LIN {X 0,Y 196.007,Z 648.874,A -85,B 0,C 180,E1 -19663.155,E2 -19663.155} C_VEL
LIN {X 0,Y 201.591,Z 629.624,A -85,B 0,C 180,E1 -19666.019,E2 -19666.019} C_VEL
LIN {X 0,Y 207.04,Z 608.516,A -85,B 0,C 180,E1 -19668.466,E2 -19668.466} C_VEL
LIN {X 0,Y 211.706,Z 587.34,A -85,B 0,C 180,E1 -19670.34,E2 -19670.34} C_VEL
LIN {X 0,Y 215.64,Z 565.396,A -85,B 0,C 180,E1 -19671.754,E2 -19671.754} C_VEL
LIN {X 0,Y 234.928,Z 427.617,A -85,B 0,C 180,E1 -19677.857,E2 -19677.857} C_VEL
LIN {X 0,Y 233.125,Z 424.133,A -85,B 0,C 180,E1 -19678.519,E2 -19678.519} C_VEL
LIN {X 0,Y 230.769,Z 425.807,A -85,B 0,C 180,E1 -19678.936,E2 -19678.936} C_VEL
LIN {X 0,Y 225.246,Z 433.176,A -85,B 0,C 180,E1 -19679.67,E2 -19679.67} C_VEL
LIN {X 0,Y 221.567,Z 436.319,A -85,B 0,C 180,E1 -19680.31,E2 -19680.31} C_VEL
LIN {X 0,Y 219.541,Z 437.961,A -85,B 0,C 180,E1 -19680.833,E2 -19680.833} C_VEL
LIN {X 0,Y 218.156,Z 442.528,A -85,B 0,C 180,E1 -19681.53,E2 -19681.53} C_VEL
LIN {X 0,Y 209.499,Z 487.735,A -85,B 0,C 180,E1 -19687.301,E2 -19687.301} C_VEL
LIN {X 0,Y 210.664,Z 518.818,A -85,B 0,C 180,E1 -19689.081,E2 -19689.081} C_VEL
LIN {X 0,Y 202.963,Z 633.554,A -85,B 0,C 180,E1 -19692.805,E2 -19692.805} C_VEL
LIN {X 0,Y 200.899,Z 650.257,A -85,B 0,C 180,E1 -19693.856,E2 -19693.856} C_VEL
LIN {X 0,Y 198.235,Z 665.159,A -85,B 0,C 180,E1 -19695.24,E2 -19695.24} C_VEL
LIN {X 0,Y 194.818,Z 679.656,A -85,B 0,C 180,E1 -19697.097,E2 -19697.097} C_VEL
LIN {X 0,Y 190.653,Z 694.187,A -85,B 0,C 180,E1 -19699.573,E2 -19699.573} C_VEL
LIN {X 0,Y 186.361,Z 706.922,A -85,B 0,C 180,E1 -19702.444,E2 -19702.444} C_VEL
LIN {X 0,Y 181.968,Z 718.732,A -85,B 0,C 180,E1 -19705.9,E2 -19705.9} C_VEL
LIN {X 0,Y 177.982,Z 728.651,A -85,B 0,C 180,E1 -19709.691,E2 -19709.691} C_VEL
LIN {X 0,Y 174.23,Z 737.787,A -85,B 0,C 180,E1 -19714.275,E2 -19714.275} C_VEL
LIN {X 0,Y 171.426,Z 744.822,A -85,B 0,C 180,E1 -19719.057,E2 -19719.057} C_VEL
LIN {X 0,Y 169.483,Z 750.379,A -85,B 0,C 180,E1 -19724.342,E2 -19724.342} C_VEL
LIN {X 0,Y 168.571,Z 753.881,A -85,B 0,C 180,E1 -19729.419,E2 -19729.419} C_VEL
LIN {X 0,Y 168.319,Z 755.89,A -85,B 0,C 180,E1 -19734.941,E2 -19734.941} C_VEL
LIN {X 0,Y 168.642,Z 756.21,A -85,B 0,C 180,E1 -19740.257,E2 -19740.257} C_VEL
LIN {X 0,Y 169.762,Z 754.819,A -85,B 0,C 180,E1 -19745.663,E2 -19745.663} C_VEL
LIN {X 0,Y 172.008,Z 751.682,A -85,B 0,C 180,E1 -19751.055,E2 -19751.055} C_VEL
LIN {X 0,Y 175.241,Z 747.035,A -85,B 0,C 180,E1 -19755.959,E2 -19755.959} C_VEL
LIN {X 0,Y 179.593,Z 740.487,A -85,B 0,C 180,E1 -19760.696,E2 -19760.696} C_VEL
LIN {X 0,Y 184.754,Z 732.288,A -85,B 0,C 180,E1 -19764.993,E2 -19764.993} C_VEL
LIN {X 0,Y 190.458,Z 722.323,A -85,B 0,C 180,E1 -19768.831,E2 -19768.831} C_VEL
LIN {X 0,Y 196.127,Z 711.358,A -85,B 0,C 180,E1 -19772.028,E2 -19772.028} C_VEL
LIN {X 0,Y 201.673,Z 698.951,A -85,B 0,C 180,E1 -19774.761,E2 -19774.761} C_VEL
LIN {X 0,Y 206.822,Z 685.498,A -85,B 0,C 180,E1 -19777.021,E2 -19777.021} C_VEL
LIN {X 0,Y 211.423,Z 670.576,A -85,B 0,C 180,E1 -19778.882,E2 -19778.882} C_VEL
LIN {X 0,Y 214.892,Z 656.116,A -85,B 0,C 180,E1 -19780.217,E2 -19780.217} C_VEL
LIN {X 0,Y 217.57,Z 640.183,A -85,B 0,C 180,E1 -19781.237,E2 -19781.237} C_VEL
LIN {X 0,Y 219.391,Z 621.388,A -85,B 0,C 180,E1 -19781.962,E2 -19781.962} C_VEL
LIN {X 0,Y 227.565,Z 519.665,A -85,B 0,C 180,E1 -19784.999,E2 -19784.999} C_VEL
LIN {X 0,Y 226.964,Z 491.665,A -85,B 0,C 180,E1 -19787.015,E2 -19787.015} C_VEL
LIN {X 0,Y 227.705,Z 486.476,A -85,B 0,C 180,E1 -19787.574,E2 -19787.574} C_VEL
LIN {X 0,Y 238.01,Z 442.856,A -85,B 0,C 180,E1 -19792.88,E2 -19792.88} C_VEL
LIN {X 0,Y 238.558,Z 440.651,A -85,B 0,C 180,E1 -19793.146,E2 -19793.146} C_VEL
LIN {X 0,Y 239.044,Z 437.189,A -85,B 0,C 180,E1 -19793.775,E2 -19793.775} C_VEL
LIN {X 0,Y 238.564,Z 433.691,A -85,B 0,C 180,E1 -19794.923,E2 -19794.923} C_VEL
LIN {X 0,Y 236.422,Z 427.479,A -85,B 0,C 180,E1 -19797.96,E2 -19797.96} C_VEL
LIN {X 0,Y 235.366,Z 419.825,A -85,B 0,C 180,E1 -19801.46,E2 -19801.46} C_VEL
LIN {X 0,Y 234.261,Z 414.19,A -85,B 0,C 180,E1 -19804.896,E2 -19804.896} C_VEL
LIN {X 0,Y 233.64,Z 409.636,A -85,B 0,C 180,E1 -19808.698,E2 -19808.698} C_VEL
LIN {X 0,Y 233.642,Z 406.373,A -85,B 0,C 180,E1 -19813.36,E2 -19813.36} C_VEL
LIN {X 0,Y 233.888,Z 406.188,A -85,B 0,C 180,E1 -19817.411,E2 -19817.411} C_VEL
LIN {X 0,Y 233.923,Z 406.605,A -85,B 0,C 180,E1 -19817.923,E2 -19817.923} C_VEL
LIN {X 0,Y 231.401,Z 422.323,A -85,B 0,C 180,E1 -19823.656,E2 -19823.656} C_VEL
LIN {X 0,Y 231.464,Z 426.766,A -85,B 0,C 180,E1 -19825.164,E2 -19825.164} C_VEL
LIN {X 0,Y 234.206,Z 432.58,A -85,B 0,C 180,E1 -19826.234,E2 -19826.234} C_VEL
LIN {X 0,Y 214.117,Z 574.365,A -85,B 0,C 180,E1 -19832.298,E2 -19832.298} C_VEL
LIN {X 0,Y 209.776,Z 596.826,A -85,B 0,C 180,E1 -19833.73,E2 -19833.73} C_VEL
LIN {X 0,Y 204.359,Z 619.531,A -85,B 0,C 180,E1 -19835.697,E2 -19835.697} C_VEL
LIN {X 0,Y 203.513,Z 624.212,A -85,B 0,C 180,E1 -19836.005,E2 -19836.005} C_VEL
LIN {X 0,Y 201.91,Z 648.108,A -85,B 0,C 180,E1 -19837.239,E2 -19837.239} C_VEL
LIN {X 0,Y 200,Z 662.648,A -85,B 0,C 180,E1 -19838.353,E2 -19838.353} C_VEL
LIN {X 0,Y 197.204,Z 676.915,A -85,B 0,C 180,E1 -19839.82,E2 -19839.82} C_VEL
LIN {X 0,Y 193.529,Z 691.091,A -85,B 0,C 180,E1 -19841.713,E2 -19841.713} C_VEL
LIN {X 0,Y 188.844,Z 705.51,A -85,B 0,C 180,E1 -19844.24,E2 -19844.24} C_VEL
LIN {X 0,Y 183.859,Z 718.529,A -85,B 0,C 180,E1 -19847.18,E2 -19847.18} C_VEL
LIN {X 0,Y 178.555,Z 730.688,A -85,B 0,C 180,E1 -19850.75,E2 -19850.75} C_VEL
LIN {X 0,Y 173.494,Z 741.383,A -85,B 0,C 180,E1 -19854.814,E2 -19854.814} C_VEL
LIN {X 0,Y 168.92,Z 750.58,A -85,B 0,C 180,E1 -19859.404,E2 -19859.404} C_VEL
LIN {X 0,Y 164.889,Z 758.8,A -85,B 0,C 180,E1 -19864.888,E2 -19864.888} C_VEL
LIN {X 0,Y 162.145,Z 764.84,A -85,B 0,C 180,E1 -19870.554,E2 -19870.554} C_VEL
LIN {X 0,Y 160.629,Z 769.021,A -85,B 0,C 180,E1 -19876.322,E2 -19876.322} C_VEL
LIN {X 0,Y 160.192,Z 771.404,A -85,B 0,C 180,E1 -19882.111,E2 -19882.111} C_VEL
LIN {X 0,Y 160.319,Z 772.033,A -85,B 0,C 180,E1 -19887.502,E2 -19887.502} C_VEL
LIN {X 0,Y 160.369,Z 771.303,A -85,B 0,C 180,E1 -19892.148,E2 -19892.148} C_VEL
LIN {X 0,Y 160.352,Z 768.92,A -85,B 0,C 180,E1 -19897.888,E2 -19897.888} C_VEL
LIN {X 0,Y 160.947,Z 769.601,A -85,B 0,C 180,E1 -19905.497,E2 -19905.497} C_VEL
LIN {X 0,Y 164.172,Z 768.537,A -85,B 0,C 180,E1 -19913.705,E2 -19913.705} C_VEL
LIN {X 0,Y 171.188,Z 765.587,A -85,B 0,C 180,E1 -19922.126,E2 -19922.126} C_VEL
LIN {X 0,Y 183.295,Z 760.405,A -85,B 0,C 180,E1 -19930.48,E2 -19930.48} C_VEL
LIN {X 0,Y 199.447,Z 753.565,A -85,B 0,C 180,E1 -19937.475,E2 -19937.475} C_VEL
LIN {X 0,Y 201.156,Z 752.825,A -85,B 0,C 180,E1 -19938.142,E2 -19938.142} C_VEL
LIN {X 0,Y 185.881,Z 756.616,A -85,B 0,C 180,E1 -19944.485,E2 -19944.485} C_VEL
LIN {X 0,Y 174.097,Z 758.634,A -85,B 0,C 180,E1 -19951.906,E2 -19951.906} C_VEL
LIN {X 0,Y 166.488,Z 758.702,A -85,B 0,C 180,E1 -19959.616,E2 -19959.616} C_VEL
LIN {X 0,Y 162.328,Z 757.034,A -85,B 0,C 180,E1 -19967.19,E2 -19967.19} C_VEL
LIN {X 0,Y 160.621,Z 753.914,A -85,B 0,C 180,E1 -19974.285,E2 -19974.285} C_VEL
LIN {X 0,Y 160.227,Z 749.933,A -85,B 0,C 180,E1 -19980.359,E2 -19980.359} C_VEL
LIN {X 0,Y 160.288,Z 744.773,A -85,B 0,C 180,E1 -19986.089,E2 -19986.089} C_VEL
LIN {X 0,Y 161.003,Z 737.672,A -85,B 0,C 180,E1 -19992.191,E2 -19992.191} C_VEL
LIN {X 0,Y 162.736,Z 728.688,A -85,B 0,C 180,E1 -19998.262,E2 -19998.262} C_VEL
LIN {X 0,Y 165.518,Z 718.279,A -85,B 0,C 180,E1 -20003.876,E2 -20003.876} C_VEL
LIN {X 0,Y 169.491,Z 705.708,A -85,B 0,C 180,E1 -20009.318,E2 -20009.318} C_VEL
LIN {X 0,Y 174.318,Z 691.587,A -85,B 0,C 180,E1 -20014.204,E2 -20014.204} C_VEL
LIN {X 0,Y 179.96,Z 675.353,A -85,B 0,C 180,E1 -20018.688,E2 -20018.688} C_VEL
LIN {X 0,Y 185.561,Z 658.707,A -85,B 0,C 180,E1 -20022.342,E2 -20022.342} C_VEL
LIN {X 0,Y 191.569,Z 639.598,A -85,B 0,C 180,E1 -20025.649,E2 -20025.649} C_VEL
LIN {X 0,Y 197.398,Z 619.056,A -85,B 0,C 180,E1 -20028.426,E2 -20028.426} C_VEL
LIN {X 0,Y 202.545,Z 598.322,A -85,B 0,C 180,E1 -20030.586,E2 -20030.586} C_VEL
LIN {X 0,Y 207.089,Z 576.326,A -85,B 0,C 180,E1 -20032.301,E2 -20032.301} C_VEL
LIN {X 0,Y 211.001,Z 551.851,A -85,B 0,C 180,E1 -20033.646,E2 -20033.646} C_VEL
LIN {X 0,Y 227.233,Z 440.079,A -85,B 0,C 180,E1 -20038.675,E2 -20038.675} C_VEL
LIN {X 0,Y 222.58,Z 443.633,A -85,B 0,C 180,E1 -20039.492,E2 -20039.492} C_VEL
LIN {X 0,Y 221.414,Z 444.853,A -85,B 0,C 180,E1 -20039.67,E2 -20039.67} C_VEL
LIN {X 0,Y 216.084,Z 451.918,A -85,B 0,C 180,E1 -20040.389,E2 -20040.389} C_VEL
LIN {X 0,Y 212.316,Z 455.133,A -85,B 0,C 180,E1 -20041.058,E2 -20041.058} C_VEL
LIN {X 0,Y 210.266,Z 456.816,A -85,B 0,C 180,E1 -20041.604,E2 -20041.604} C_VEL
LIN {X 0,Y 208.844,Z 461.49,A -85,B 0,C 180,E1 -20042.326,E2 -20042.326} C_VEL
LIN {X 0,Y 203.614,Z 488.758,A -85,B 0,C 180,E1 -20045.822,E2 -20045.822} C_VEL
LIN {X 0,Y 204.632,Z 519.551,A -85,B 0,C 180,E1 -20047.637,E2 -20047.637} C_VEL
LIN {X 0,Y 196.623,Z 633.934,A -85,B 0,C 180,E1 -20051.409,E2 -20051.409} C_VEL
LIN {X 0,Y 194.482,Z 650.561,A -85,B 0,C 180,E1 -20052.475,E2 -20052.475} C_VEL
LIN {X 0,Y 191.599,Z 665.988,A -85,B 0,C 180,E1 -20053.941,E2 -20053.941} C_VEL
LIN {X 0,Y 187.788,Z 681.269,A -85,B 0,C 180,E1 -20055.977,E2 -20055.977} C_VEL
LIN {X 0,Y 183.461,Z 695.537,A -85,B 0,C 180,E1 -20058.523,E2 -20058.523} C_VEL
LIN {X 0,Y 178.786,Z 708.651,A -85,B 0,C 180,E1 -20061.636,E2 -20061.636} C_VEL
LIN {X 0,Y 174.426,Z 719.757,A -85,B 0,C 180,E1 -20065.064,E2 -20065.064} C_VEL
LIN {X 0,Y 169.976,Z 730.229,A -85,B 0,C 180,E1 -20069.322,E2 -20069.322} C_VEL
LIN {X 0,Y 166.35,Z 738.634,A -85,B 0,C 180,E1 -20073.816,E2 -20073.816} C_VEL
LIN {X 0,Y 163.459,Z 745.511,A -85,B 0,C 180,E1 -20078.792,E2 -20078.792} C_VEL
LIN {X 0,Y 161.462,Z 750.998,A -85,B 0,C 180,E1 -20084.337,E2 -20084.337} C_VEL
LIN {X 0,Y 160.513,Z 754.566,A -85,B 0,C 180,E1 -20090.031,E2 -20090.031} C_VEL
LIN {X 0,Y 160.333,Z 756.348,A -85,B 0,C 180,E1 -20095.482,E2 -20095.482} C_VEL
LIN {X 0,Y 160.754,Z 756.579,A -85,B 0,C 180,E1 -20101.076,E2 -20101.076} C_VEL
LIN {X 0,Y 162.224,Z 754.933,A -85,B 0,C 180,E1 -20107.153,E2 -20107.153} C_VEL
LIN {X 0,Y 164.898,Z 751.567,A -85,B 0,C 180,E1 -20112.802,E2 -20112.802} C_VEL
LIN {X 0,Y 168.893,Z 746.228,A -85,B 0,C 180,E1 -20118.232,E2 -20118.232} C_VEL
LIN {X 0,Y 173.835,Z 739.315,A -85,B 0,C 180,E1 -20123.075,E2 -20123.075} C_VEL
LIN {X 0,Y 179.748,Z 730.328,A -85,B 0,C 180,E1 -20127.556,E2 -20127.556} C_VEL
LIN {X 0,Y 185.805,Z 720.142,A -85,B 0,C 180,E1 -20131.291,E2 -20131.291} C_VEL
LIN {X 0,Y 192.09,Z 708.2,A -85,B 0,C 180,E1 -20134.56,E2 -20134.56} C_VEL
LIN {X 0,Y 197.59,Z 696.12,A -85,B 0,C 180,E1 -20137.067,E2 -20137.067} C_VEL
LIN {X 0,Y 203.058,Z 681.742,A -85,B 0,C 180,E1 -20139.308,E2 -20139.308} C_VEL
LIN {X 0,Y 207.513,Z 667.094,A -85,B 0,C 180,E1 -20141.001,E2 -20141.001} C_VEL
LIN {X 0,Y 211.23,Z 650.563,A -85,B 0,C 180,E1 -20142.364,E2 -20142.364} C_VEL
LIN {X 0,Y 213.59,Z 634.571,A -85,B 0,C 180,E1 -20143.234,E2 -20143.234} C_VEL
LIN {X 0,Y 223.224,Z 520.734,A -85,B 0,C 180,E1 -20146.695,E2 -20146.695} C_VEL
LIN {X 0,Y 222.906,Z 493.056,A -85,B 0,C 180,E1 -20148.747,E2 -20148.747} C_VEL
LIN {X 0,Y 223.234,Z 488.794,A -85,B 0,C 180,E1 -20149.156,E2 -20149.156} C_VEL
LIN {X 0,Y 233.54,Z 447.232,A -85,B 0,C 180,E1 -20154.225,E2 -20154.225} C_VEL
LIN {X 0,Y 237.089,Z 432.81,A -85,B 0,C 180,E1 -20156.009,E2 -20156.009} C_VEL
LIN {X 0,Y 236.422,Z 427.479,A -85,B 0,C 180,E1 -20157.96,E2 -20157.96} C_VEL
LIN {X 0,Y 235.623,Z 424.837,A -85,B 0,C 180,E1 -20159.425,E2 -20159.425} C_VEL
LIN {X 0,Y 233.667,Z 422.928,A -85,B 0,C 180,E1 -20161.79,E2 -20161.79} C_VEL
LIN {X 0,Y 231.182,Z 421.007,A -85,B 0,C 180,E1 -20165.355,E2 -20165.355} C_VEL
LIN {X 0,Y 230.926,Z 419.801,A -85,B 0,C 180,E1 -20166.437,E2 -20166.437} C_VEL
LIN {X 0,Y 230.46,Z 416.606,A -85,B 0,C 180,E1 -20169.488,E2 -20169.488} C_VEL
LIN {X 0,Y 230.78,Z 413.806,A -85,B 0,C 180,E1 -20173.785,E2 -20173.785} C_VEL
LIN {X 0,Y 231.018,Z 413.815,A -85,B 0,C 180,E1 -20177.245,E2 -20177.245} C_VEL
LIN {X 0,Y 228.173,Z 430.939,A -85,B 0,C 180,E1 -20183.5,E2 -20183.5} C_VEL
LIN {X 0,Y 228.012,Z 435.468,A -85,B 0,C 180,E1 -20184.971,E2 -20184.971} C_VEL
LIN {X 0,Y 207.408,Z 574.805,A -85,B 0,C 180,E1 -20191.105,E2 -20191.105} C_VEL
LIN {X 0,Y 202.897,Z 597.264,A -85,B 0,C 180,E1 -20192.583,E2 -20192.583} C_VEL
LIN {X 0,Y 201.248,Z 605.535,A -85,B 0,C 180,E1 -20193.136,E2 -20193.136} C_VEL
LIN {X 0,Y 200.055,Z 621.802,A -85,B 0,C 180,E1 -20193.871,E2 -20193.871} C_VEL
LIN {X 0,Y 199.017,Z 637.587,A -85,B 0,C 180,E1 -20194.64,E2 -20194.64} C_VEL
LIN {X 0,Y 197.793,Z 650.252,A -85,B 0,C 180,E1 -20195.36,E2 -20195.36} C_VEL
LIN {X 0,Y 195.668,Z 663.933,A -85,B 0,C 180,E1 -20196.44,E2 -20196.44} C_VEL
LIN {X 0,Y 192.609,Z 677.955,A -85,B 0,C 180,E1 -20197.909,E2 -20197.909} C_VEL
LIN {X 0,Y 188.65,Z 691.693,A -85,B 0,C 180,E1 -20199.786,E2 -20199.786} C_VEL
LIN {X 0,Y 183.485,Z 706.278,A -85,B 0,C 180,E1 -20202.398,E2 -20202.398} C_VEL
LIN {X 0,Y 178.044,Z 719.249,A -85,B 0,C 180,E1 -20205.42,E2 -20205.42} C_VEL
LIN {X 0,Y 172.357,Z 731.173,A -85,B 0,C 180,E1 -20209.046,E2 -20209.046} C_VEL
LIN {X 0,Y 166.901,Z 741.673,A -85,B 0,C 180,E1 -20213.202,E2 -20213.202} C_VEL
LIN {X 0,Y 161.621,Z 751.27,A -85,B 0,C 180,E1 -20218.28,E2 -20218.28} C_VEL
LIN {X 0,Y 157.511,Z 758.77,A -85,B 0,C 180,E1 -20223.623,E2 -20223.623} C_VEL
LIN {X 0,Y 154.463,Z 764.695,A -85,B 0,C 180,E1 -20229.545,E2 -20229.545} C_VEL
LIN {X 0,Y 152.725,Z 768.827,A -85,B 0,C 180,E1 -20235.674,E2 -20235.674} C_VEL
LIN {X 0,Y 152.201,Z 771.06,A -85,B 0,C 180,E1 -20241.694,E2 -20241.694} C_VEL
LIN {X 0,Y 152.323,Z 771.623,A -85,B 0,C 180,E1 -20247.371,E2 -20247.371} C_VEL
LIN {X 0,Y 152.378,Z 770.824,A -85,B 0,C 180,E1 -20252.26,E2 -20252.26} C_VEL
LIN {X 0,Y 152.369,Z 768.382,A -85,B 0,C 180,E1 -20257.925,E2 -20257.925} C_VEL
LIN {X 0,Y 152.403,Z 768.051,A -85,B 0,C 180,E1 -20259.063,E2 -20259.063} C_VEL
LIN {X 0,Y 153.327,Z 768.816,A -85,B 0,C 180,E1 -20267.069,E2 -20267.069} C_VEL
LIN {X 0,Y 157.422,Z 767.916,A -85,B 0,C 180,E1 -20275.996,E2 -20275.996} C_VEL
LIN {X 0,Y 166.294,Z 764.952,A -85,B 0,C 180,E1 -20285.259,E2 -20285.259} C_VEL
LIN {X 0,Y 179.981,Z 760.058,A -85,B 0,C 180,E1 -20293.544,E2 -20293.544} C_VEL
LIN {X 0,Y 190.979,Z 756.033,A -85,B 0,C 180,E1 -20298.205,E2 -20298.205} C_VEL
LIN {X 0,Y 175.669,Z 758.775,A -85,B 0,C 180,E1 -20305.051,E2 -20305.051} C_VEL
LIN {X 0,Y 164.759,Z 759.68,A -85,B 0,C 180,E1 -20312.536,E2 -20312.536} C_VEL
LIN {X 0,Y 157.483,Z 758.803,A -85,B 0,C 180,E1 -20320.724,E2 -20320.724} C_VEL
LIN {X 0,Y 153.749,Z 756.259,A -85,B 0,C 180,E1 -20328.751,E2 -20328.751} C_VEL
LIN {X 0,Y 152.428,Z 752.31,A -85,B 0,C 180,E1 -20336.24,E2 -20336.24} C_VEL
LIN {X 0,Y 152.211,Z 747.873,A -85,B 0,C 180,E1 -20342.26,E2 -20342.26} C_VEL
LIN {X 0,Y 152.462,Z 741.959,A -85,B 0,C 180,E1 -20348.297,E2 -20348.297} C_VEL
LIN {X 0,Y 153.556,Z 733.994,A -85,B 0,C 180,E1 -20354.712,E2 -20354.712} C_VEL
LIN {X 0,Y 155.863,Z 724.042,A -85,B 0,C 180,E1 -20361.055,E2 -20361.055} C_VEL
LIN {X 0,Y 159.422,Z 712.205,A -85,B 0,C 180,E1 -20367.045,E2 -20367.045} C_VEL
LIN {X 0,Y 164.001,Z 698.806,A -85,B 0,C 180,E1 -20372.448,E2 -20372.448} C_VEL
LIN {X 0,Y 169.34,Z 683.884,A -85,B 0,C 180,E1 -20377.245,E2 -20377.245} C_VEL
LIN {X 0,Y 175.192,Z 667.429,A -85,B 0,C 180,E1 -20381.457,E2 -20381.457} C_VEL
LIN {X 0,Y 181.263,Z 649.43,A -85,B 0,C 180,E1 -20385.081,E2 -20385.081} C_VEL
LIN {X 0,Y 187.216,Z 630.282,A -85,B 0,C 180,E1 -20388.116,E2 -20388.116} C_VEL
LIN {X 0,Y 193.011,Z 609.33,A -85,B 0,C 180,E1 -20390.692,E2 -20390.692} C_VEL
LIN {X 0,Y 198.029,Z 588.042,A -85,B 0,C 180,E1 -20392.679,E2 -20392.679} C_VEL
LIN {X 0,Y 202.33,Z 565.771,A -85,B 0,C 180,E1 -20394.195,E2 -20394.195} C_VEL
LIN {X 0,Y 218.439,Z 458.466,A -85,B 0,C 180,E1 -20399.293,E2 -20399.293} C_VEL
LIN {X 0,Y 213.978,Z 462.059,A -85,B 0,C 180,E1 -20400.076,E2 -20400.076} C_VEL
LIN {X 0,Y 212.508,Z 463.195,A -85,B 0,C 180,E1 -20400.339,E2 -20400.339} C_VEL
LIN {X 0,Y 207.004,Z 470.589,A -85,B 0,C 180,E1 -20401.075,E2 -20401.075} C_VEL
LIN {X 0,Y 203.137,Z 473.924,A -85,B 0,C 180,E1 -20401.772,E2 -20401.772} C_VEL
LIN {X 0,Y 201.131,Z 475.381,A -85,B 0,C 180,E1 -20402.299,E2 -20402.299} C_VEL
LIN {X 0,Y 199.828,Z 478.864,A -85,B 0,C 180,E1 -20402.911,E2 -20402.911} C_VEL
LIN {X 0,Y 197.861,Z 489.188,A -85,B 0,C 180,E1 -20404.218,E2 -20404.218} C_VEL
LIN {X 0,Y 198.705,Z 520.426,A -85,B 0,C 180,E1 -20406.116,E2 -20406.116} C_VEL
LIN {X 0,Y 190.39,Z 634.283,A -85,B 0,C 180,E1 -20409.927,E2 -20409.927} C_VEL
LIN {X 0,Y 188.148,Z 650.98,A -85,B 0,C 180,E1 -20411.015,E2 -20411.015} C_VEL
LIN {X 0,Y 185.065,Z 666.733,A -85,B 0,C 180,E1 -20412.548,E2 -20412.548} C_VEL
LIN {X 0,Y 181.093,Z 681.937,A -85,B 0,C 180,E1 -20414.628,E2 -20414.628} C_VEL
LIN {X 0,Y 176.819,Z 695.455,A -85,B 0,C 180,E1 -20417.09,E2 -20417.09} C_VEL
LIN {X 0,Y 171.909,Z 708.656,A -85,B 0,C 180,E1 -20420.286,E2 -20420.286} C_VEL
LIN {X 0,Y 167.314,Z 719.842,A -85,B 0,C 180,E1 -20423.821,E2 -20423.821} C_VEL
LIN {X 0,Y 162.608,Z 730.379,A -85,B 0,C 180,E1 -20428.234,E2 -20428.234} C_VEL
LIN {X 0,Y 158.779,Z 738.788,A -85,B 0,C 180,E1 -20432.884,E2 -20432.884} C_VEL
LIN {X 0,Y 155.602,Z 745.937,A -85,B 0,C 180,E1 -20438.274,E2 -20438.274} C_VEL
LIN {X 0,Y 153.529,Z 751.319,A -85,B 0,C 180,E1 -20443.977,E2 -20443.977} C_VEL
LIN {X 0,Y 152.525,Z 754.902,A -85,B 0,C 180,E1 -20449.926,E2 -20449.926} C_VEL
LIN {X 0,Y 152.349,Z 756.776,A -85,B 0,C 180,E1 -20455.954,E2 -20455.954} C_VEL
LIN {X 0,Y 152.859,Z 756.971,A -85,B 0,C 180,E1 -20461.749,E2 -20461.749} C_VEL
LIN {X 0,Y 154.466,Z 755.389,A -85,B 0,C 180,E1 -20467.942,E2 -20467.942} C_VEL
LIN {X 0,Y 157.379,Z 752.102,A -85,B 0,C 180,E1 -20473.822,E2 -20473.822} C_VEL
LIN {X 0,Y 161.744,Z 746.766,A -85,B 0,C 180,E1 -20479.526,E2 -20479.526} C_VEL
LIN {X 0,Y 167.015,Z 739.953,A -85,B 0,C 180,E1 -20484.499,E2 -20484.499} C_VEL
LIN {X 0,Y 173.311,Z 731.031,A -85,B 0,C 180,E1 -20489.104,E2 -20489.104} C_VEL
LIN {X 0,Y 179.697,Z 721.022,A -85,B 0,C 180,E1 -20492.897,E2 -20492.897} C_VEL
LIN {X 0,Y 185.971,Z 709.823,A -85,B 0,C 180,E1 -20496.053,E2 -20496.053} C_VEL
LIN {X 0,Y 192.047,Z 697.314,A -85,B 0,C 180,E1 -20498.727,E2 -20498.727} C_VEL
LIN {X 0,Y 197.355,Z 684.211,A -85,B 0,C 180,E1 -20500.829,E2 -20500.829} C_VEL
LIN {X 0,Y 202.206,Z 669.444,A -85,B 0,C 180,E1 -20502.606,E2 -20502.606} C_VEL
LIN {X 0,Y 205.999,Z 654.08,A -85,B 0,C 180,E1 -20503.939,E2 -20503.939} C_VEL
LIN {X 0,Y 208.829,Z 637.258,A -85,B 0,C 180,E1 -20504.928,E2 -20504.928} C_VEL
LIN {X 0,Y 213.042,Z 590.682,A -85,B 0,C 180,E1 -20506.414,E2 -20506.414} C_VEL
LIN {X 0,Y 219.172,Z 521.821,A -85,B 0,C 180,E1 -20508.47,E2 -20508.47} C_VEL
LIN {X 0,Y 219.13,Z 494.343,A -85,B 0,C 180,E1 -20510.561,E2 -20510.561} C_VEL
LIN {X 0,Y 219.29,Z 489.996,A -85,B 0,C 180,E1 -20510.949,E2 -20510.949} C_VEL
LIN {X 0,Y 230.062,Z 448.378,A -85,B 0,C 180,E1 -20516.012,E2 -20516.012} C_VEL
LIN {X 0,Y 232.935,Z 437.369,A -85,B 0,C 180,E1 -20517.354,E2 -20517.354} C_VEL
LIN {X 0,Y 232.182,Z 429.752,A -85,B 0,C 180,E1 -20520.493,E2 -20520.493} C_VEL
LIN {X 0,Y 231.38,Z 424.088,A -85,B 0,C 180,E1 -20523.479,E2 -20523.479} C_VEL
LIN {X 0,Y 230.926,Z 419.801,A -85,B 0,C 180,E1 -20526.437,E2 -20526.437} C_VEL
LIN {X 0,Y 230.574,Z 418.534,A -85,B 0,C 180,E1 -20528.047,E2 -20528.047} C_VEL
LIN {X 0,Y 229.588,Z 418.914,A -85,B 0,C 180,E1 -20530.39,E2 -20530.39} C_VEL
LIN {X 0,Y 228.041,Z 421.125,A -85,B 0,C 180,E1 -20534.624,E2 -20534.624} C_VEL
LIN {X 0,Y 227.979,Z 421.154,A -85,B 0,C 180,E1 -20535.341,E2 -20535.341} C_VEL
LIN {X 0,Y 228.094,Z 421.22,A -85,B 0,C 180,E1 -20536.619,E2 -20536.619} C_VEL
LIN {X 0,Y 225.005,Z 438.69,A -85,B 0,C 180,E1 -20543.019,E2 -20543.019} C_VEL
LIN {X 0,Y 224.901,Z 439.395,A -85,B 0,C 180,E1 -20543.205,E2 -20543.205} C_VEL
LIN {X 0,Y 217.624,Z 464.437,A -85,B 0,C 180,E1 -20544.753,E2 -20544.753} C_VEL
LIN {X 0,Y 200.394,Z 578.791,A -85,B 0,C 180,E1 -20549.941,E2 -20549.941} C_VEL
LIN {X 0,Y 198.399,Z 601.252,A -85,B 0,C 180,E1 -20550.827,E2 -20550.827} C_VEL
LIN {X 0,Y 196.659,Z 622.745,A -85,B 0,C 180,E1 -20551.794,E2 -20551.794} C_VEL
LIN {X 0,Y 194.44,Z 647.901,A -85,B 0,C 180,E1 -20553.058,E2 -20553.058} C_VEL
LIN {X 0,Y 191.865,Z 663.877,A -85,B 0,C 180,E1 -20554.298,E2 -20554.298} C_VEL
LIN {X 0,Y 188.236,Z 678.98,A -85,B 0,C 180,E1 -20555.907,E2 -20555.907} C_VEL
LIN {X 0,Y 183.539,Z 693.743,A -85,B 0,C 180,E1 -20557.993,E2 -20557.993} C_VEL
LIN {X 0,Y 178.346,Z 707.121,A -85,B 0,C 180,E1 -20560.45,E2 -20560.45} C_VEL
LIN {X 0,Y 172.064,Z 720.719,A -85,B 0,C 180,E1 -20563.748,E2 -20563.748} C_VEL
LIN {X 0,Y 165.86,Z 732.583,A -85,B 0,C 180,E1 -20567.538,E2 -20567.538} C_VEL
LIN {X 0,Y 159.63,Z 743.349,A -85,B 0,C 180,E1 -20572.138,E2 -20572.138} C_VEL
LIN {X 0,Y 154.392,Z 751.973,A -85,B 0,C 180,E1 -20577.049,E2 -20577.049} C_VEL
LIN {X 0,Y 149.964,Z 759.156,A -85,B 0,C 180,E1 -20582.615,E2 -20582.615} C_VEL
LIN {X 0,Y 146.667,Z 764.871,A -85,B 0,C 180,E1 -20588.824,E2 -20588.824} C_VEL
LIN {X 0,Y 144.791,Z 768.714,A -85,B 0,C 180,E1 -20595.201,E2 -20595.201} C_VEL
LIN {X 0,Y 144.205,Z 770.801,A -85,B 0,C 180,E1 -20601.632,E2 -20601.632} C_VEL
LIN {X 0,Y 144.327,Z 771.212,A -85,B 0,C 180,E1 -20607.225,E2 -20607.225} C_VEL
LIN {X 0,Y 144.394,Z 770.455,A -85,B 0,C 180,E1 -20611.988,E2 -20611.988} C_VEL
LIN {X 0,Y 144.368,Z 768.226,A -85,B 0,C 180,E1 -20617.566,E2 -20617.566} C_VEL
LIN {X 0,Y 144.49,Z 767.034,A -85,B 0,C 180,E1 -20619.966,E2 -20619.966} C_VEL
LIN {X 0,Y 145.948,Z 768.02,A -85,B 0,C 180,E1 -20629.202,E2 -20629.202} C_VEL
LIN {X 0,Y 151.239,Z 767.234,A -85,B 0,C 180,E1 -20638.86,E2 -20638.86} C_VEL
LIN {X 0,Y 161.503,Z 764.512,A -85,B 0,C 180,E1 -20648.254,E2 -20648.254} C_VEL
LIN {X 0,Y 176.639,Z 760.01,A -85,B 0,C 180,E1 -20656.435,E2 -20656.435} C_VEL
LIN {X 0,Y 180.856,Z 758.644,A -85,B 0,C 180,E1 -20658.228,E2 -20658.228} C_VEL
LIN {X 0,Y 166.303,Z 760.289,A -85,B 0,C 180,E1 -20665.17,E2 -20665.17} C_VEL
LIN {X 0,Y 155.426,Z 760.26,A -85,B 0,C 180,E1 -20673.238,E2 -20673.238} C_VEL
LIN {X 0,Y 148.532,Z 758.45,A -85,B 0,C 180,E1 -20681.963,E2 -20681.963} C_VEL
LIN {X 0,Y 145.264,Z 755.031,A -85,B 0,C 180,E1 -20690.493,E2 -20690.493} C_VEL
LIN {X 0,Y 144.339,Z 750.518,A -85,B 0,C 180,E1 -20698.017,E2 -20698.017} C_VEL
LIN {X 0,Y 144.254,Z 745.363,A -85,B 0,C 180,E1 -20704.374,E2 -20704.374} C_VEL
LIN {X 0,Y 144.765,Z 738.683,A -85,B 0,C 180,E1 -20710.749,E2 -20710.749} C_VEL
LIN {X 0,Y 146.359,Z 729.797,A -85,B 0,C 180,E1 -20717.494,E2 -20717.494} C_VEL
LIN {X 0,Y 149.333,Z 718.796,A -85,B 0,C 180,E1 -20724.107,E2 -20724.107} C_VEL
LIN {X 0,Y 153.499,Z 706.229,A -85,B 0,C 180,E1 -20730.105,E2 -20730.105} C_VEL
LIN {X 0,Y 158.616,Z 692.123,A -85,B 0,C 180,E1 -20735.448,E2 -20735.448} C_VEL
LIN {X 0,Y 164.624,Z 675.94,A -85,B 0,C 180,E1 -20740.305,E2 -20740.305} C_VEL
LIN {X 0,Y 170.871,Z 658.525,A -85,B 0,C 180,E1 -20744.393,E2 -20744.393} C_VEL
LIN {X 0,Y 177.259,Z 639.518,A -85,B 0,C 180,E1 -20747.882,E2 -20747.882} C_VEL
LIN {X 0,Y 183.384,Z 619.315,A -85,B 0,C 180,E1 -20750.764,E2 -20750.764} C_VEL
LIN {X 0,Y 188.924,Z 598.368,A -85,B 0,C 180,E1 -20753.051,E2 -20753.051} C_VEL
LIN {X 0,Y 193.811,Z 576.226,A -85,B 0,C 180,E1 -20754.856,E2 -20754.856} C_VEL
LIN {X 0,Y 198.126,Z 551.12,A -85,B 0,C 180,E1 -20756.305,E2 -20756.305} C_VEL
LIN {X 0,Y 209.631,Z 476.889,A -85,B 0,C 180,E1 -20759.892,E2 -20759.892} C_VEL
LIN {X 0,Y 205.044,Z 480.699,A -85,B 0,C 180,E1 -20760.696,E2 -20760.696} C_VEL
LIN {X 0,Y 203.21,Z 482.007,A -85,B 0,C 180,E1 -20761.042,E2 -20761.042} C_VEL
LIN {X 0,Y 197.545,Z 489.63,A -85,B 0,C 180,E1 -20761.805,E2 -20761.805} C_VEL
LIN {X 0,Y 193.811,Z 493.658,A -85,B 0,C 180,E1 -20762.449,E2 -20762.449} C_VEL
LIN {X 0,Y 192.684,Z 496.1,A -85,B 0,C 180,E1 -20762.868,E2 -20762.868} C_VEL
LIN {X 0,Y 192.749,Z 509.195,A -85,B 0,C 180,E1 -20763.786,E2 -20763.786} C_VEL
LIN {X 0,Y 192.907,Z 521.389,A -85,B 0,C 180,E1 -20764.511,E2 -20764.511} C_VEL
LIN {X 0,Y 184.25,Z 634.762,A -85,B 0,C 180,E1 -20768.363,E2 -20768.363} C_VEL
LIN {X 0,Y 181.903,Z 651.472,A -85,B 0,C 180,E1 -20769.473,E2 -20769.473} C_VEL
LIN {X 0,Y 178.643,Z 667.365,A -85,B 0,C 180,E1 -20771.054,E2 -20771.054} C_VEL
LIN {X 0,Y 174.391,Z 682.892,A -85,B 0,C 180,E1 -20773.237,E2 -20773.237} C_VEL
LIN {X 0,Y 169.782,Z 696.676,A -85,B 0,C 180,E1 -20775.85,E2 -20775.85} C_VEL
LIN {X 0,Y 164.438,Z 710.307,A -85,B 0,C 180,E1 -20779.309,E2 -20779.309} C_VEL
LIN {X 0,Y 159.461,Z 721.651,A -85,B 0,C 180,E1 -20783.154,E2 -20783.154} C_VEL
LIN {X 0,Y 154.615,Z 731.945,A -85,B 0,C 180,E1 -20787.772,E2 -20787.772} C_VEL
LIN {X 0,Y 150.686,Z 740.07,A -85,B 0,C 180,E1 -20792.658,E2 -20792.658} C_VEL
LIN {X 0,Y 147.355,Z 747.278,A -85,B 0,C 180,E1 -20798.581,E2 -20798.581} C_VEL
LIN {X 0,Y 145.412,Z 752.155,A -85,B 0,C 180,E1 -20804.327,E2 -20804.327} C_VEL
LIN {X 0,Y 144.455,Z 755.672,A -85,B 0,C 180,E1 -20810.862,E2 -20810.862} C_VEL
LIN {X 0,Y 144.383,Z 757.254,A -85,B 0,C 180,E1 -20816.747,E2 -20816.747} C_VEL
LIN {X 0,Y 145.069,Z 757.297,A -85,B 0,C 180,E1 -20822.984,E2 -20822.984} C_VEL
LIN {X 0,Y 147.107,Z 755.522,A -85,B 0,C 180,E1 -20829.704,E2 -20829.704} C_VEL
LIN {X 0,Y 150.512,Z 751.971,A -85,B 0,C 180,E1 -20835.838,E2 -20835.838} C_VEL
LIN {X 0,Y 155.429,Z 746.493,A -85,B 0,C 180,E1 -20841.696,E2 -20841.696} C_VEL
LIN {X 0,Y 161.284,Z 739.378,A -85,B 0,C 180,E1 -20846.807,E2 -20846.807} C_VEL
LIN {X 0,Y 168.033,Z 730.398,A -85,B 0,C 180,E1 -20851.394,E2 -20851.394} C_VEL
LIN {X 0,Y 174.741,Z 720.288,A -85,B 0,C 180,E1 -20855.132,E2 -20855.132} C_VEL
LIN {X 0,Y 181.709,Z 708.335,A -85,B 0,C 180,E1 -20858.412,E2 -20858.412} C_VEL
LIN {X 0,Y 188.141,Z 695.233,A -85,B 0,C 180,E1 -20861.066,E2 -20861.066} C_VEL
LIN {X 0,Y 193.985,Z 680.932,A -85,B 0,C 180,E1 -20863.222,E2 -20863.222} C_VEL
LIN {X 0,Y 198.833,Z 665.791,A -85,B 0,C 180,E1 -20864.891,E2 -20864.891} C_VEL
LIN {X 0,Y 202.615,Z 649.924,A -85,B 0,C 180,E1 -20866.143,E2 -20866.143} C_VEL
LIN {X 0,Y 205.157,Z 633.142,A -85,B 0,C 180,E1 -20866.996,E2 -20866.996} C_VEL
LIN {X 0,Y 215.388,Z 522.939,A -85,B 0,C 180,E1 -20870.314,E2 -20870.314} C_VEL
LIN {X 0,Y 215.606,Z 495.453,A -85,B 0,C 180,E1 -20872.454,E2 -20872.454} C_VEL
LIN {X 0,Y 215.915,Z 490.055,A -85,B 0,C 180,E1 -20872.95,E2 -20872.95} C_VEL
LIN {X 0,Y 227.818,Z 446.411,A -85,B 0,C 180,E1 -20878.239,E2 -20878.239} C_VEL
LIN {X 0,Y 229.039,Z 441.918,A -85,B 0,C 180,E1 -20878.811,E2 -20878.811} C_VEL
LIN {X 0,Y 228.47,Z 434.651,A -85,B 0,C 180,E1 -20882.005,E2 -20882.005} C_VEL
LIN {X 0,Y 227.892,Z 428.743,A -85,B 0,C 180,E1 -20885.538,E2 -20885.538} C_VEL
LIN {X 0,Y 227.573,Z 424.262,A -85,B 0,C 180,E1 -20889.355,E2 -20889.355} C_VEL
LIN {X 0,Y 227.918,Z 421.264,A -85,B 0,C 180,E1 -20893.961,E2 -20893.961} C_VEL
LIN {X 0,Y 227.979,Z 421.154,A -85,B 0,C 180,E1 -20895.341,E2 -20895.341} C_VEL
LIN {X 0,Y 227.686,Z 422.083,A -85,B 0,C 180,E1 -20896.18,E2 -20896.18} C_VEL
LIN {X 0,Y 226.697,Z 425.422,A -85,B 0,C 180,E1 -20897.121,E2 -20897.121} C_VEL
LIN {X 0,Y 223.576,Z 435.876,A -85,B 0,C 180,E1 -20898.884,E2 -20898.884} C_VEL
LIN {X 0,Y 223.089,Z 438.023,A -85,B 0,C 180,E1 -20899.497,E2 -20899.497} C_VEL
LIN {X 0,Y 222.206,Z 443.371,A -85,B 0,C 180,E1 -20901.374,E2 -20901.374} C_VEL
LIN {X 0,Y 207.733,Z 490.679,A -85,B 0,C 180,E1 -20904.38,E2 -20904.38} C_VEL
LIN {X 0,Y 205.088,Z 506.599,A -85,B 0,C 180,E1 -20905.128,E2 -20905.128} C_VEL
LIN {X 0,Y 198.317,Z 572.607,A -85,B 0,C 180,E1 -20907.552,E2 -20907.552} C_VEL
LIN {X 0,Y 195.547,Z 601.102,A -85,B 0,C 180,E1 -20908.623,E2 -20908.623} C_VEL
LIN {X 0,Y 193.567,Z 624.291,A -85,B 0,C 180,E1 -20909.674,E2 -20909.674} C_VEL
LIN {X 0,Y 191.31,Z 647.465,A -85,B 0,C 180,E1 -20910.818,E2 -20910.818} C_VEL
LIN {X 0,Y 188.482,Z 663.492,A -85,B 0,C 180,E1 -20912.037,E2 -20912.037} C_VEL
LIN {X 0,Y 184.425,Z 679.041,A -85,B 0,C 180,E1 -20913.682,E2 -20913.682} C_VEL
LIN {X 0,Y 179.326,Z 693.956,A -85,B 0,C 180,E1 -20915.78,E2 -20915.78} C_VEL
LIN {X 0,Y 173.445,Z 707.897,A -85,B 0,C 180,E1 -20918.379,E2 -20918.379} C_VEL
LIN {X 0,Y 166.565,Z 721.606,A -85,B 0,C 180,E1 -20921.781,E2 -20921.781} C_VEL
LIN {X 0,Y 159.981,Z 733.088,A -85,B 0,C 180,E1 -20925.58,E2 -20925.58} C_VEL
LIN {X 0,Y 153.124,Z 743.911,A -85,B 0,C 180,E1 -20930.398,E2 -20930.398} C_VEL
LIN {X 0,Y 147.235,Z 752.62,A -85,B 0,C 180,E1 -20935.697,E2 -20935.697} C_VEL
LIN {X 0,Y 142.202,Z 759.961,A -85,B 0,C 180,E1 -20941.9,E2 -20941.9} C_VEL
LIN {X 0,Y 138.724,Z 765.29,A -85,B 0,C 180,E1 -20948.438,E2 -20948.438} C_VEL
LIN {X 0,Y 136.699,Z 768.974,A -85,B 0,C 180,E1 -20955.605,E2 -20955.605} C_VEL
LIN {X 0,Y 136.202,Z 770.659,A -85,B 0,C 180,E1 -20962.412,E2 -20962.412} C_VEL
LIN {X 0,Y 136.38,Z 770.694,A -85,B 0,C 180,E1 -20968.324,E2 -20968.324} C_VEL
LIN {X 0,Y 136.378,Z 769.624,A -85,B 0,C 180,E1 -20973.367,E2 -20973.367} C_VEL
LIN {X 0,Y 136.448,Z 766.979,A -85,B 0,C 180,E1 -20979.282,E2 -20979.282} C_VEL
LIN {X 0,Y 136.634,Z 766.026,A -85,B 0,C 180,E1 -20981.4,E2 -20981.4} C_VEL
LIN {X 0,Y 138.841,Z 767.204,A -85,B 0,C 180,E1 -20991.726,E2 -20991.726} C_VEL
LIN {X 0,Y 145.472,Z 766.561,A -85,B 0,C 180,E1 -21001.958,E2 -21001.958} C_VEL
LIN {X 0,Y 157.729,Z 763.951,A -85,B 0,C 180,E1 -21011.733,E2 -21011.733} C_VEL
LIN {X 0,Y 170.729,Z 760.685,A -85,B 0,C 180,E1 -21018.241,E2 -21018.241} C_VEL
LIN {X 0,Y 156.243,Z 761.337,A -85,B 0,C 180,E1 -21025.728,E2 -21025.728} C_VEL
LIN {X 0,Y 145.762,Z 760.293,A -85,B 0,C 180,E1 -21034.397,E2 -21034.397} C_VEL
LIN {X 0,Y 139.457,Z 757.48,A -85,B 0,C 180,E1 -21043.764,E2 -21043.764} C_VEL
LIN {X 0,Y 136.886,Z 753.335,A -85,B 0,C 180,E1 -21052.447,E2 -21052.447} C_VEL
LIN {X 0,Y 136.308,Z 748.658,A -85,B 0,C 180,E1 -21059.581,E2 -21059.581} C_VEL
LIN {X 0,Y 136.364,Z 742.798,A -85,B 0,C 180,E1 -21066.316,E2 -21066.316} C_VEL
LIN {X 0,Y 137.263,Z 734.901,A -85,B 0,C 180,E1 -21073.481,E2 -21073.481} C_VEL
LIN {X 0,Y 139.461,Z 725.036,A -85,B 0,C 180,E1 -21080.569,E2 -21080.569} C_VEL
LIN {X 0,Y 142.943,Z 713.689,A -85,B 0,C 180,E1 -21087.045,E2 -21087.045} C_VEL
LIN {X 0,Y 147.839,Z 700.038,A -85,B 0,C 180,E1 -21093.219,E2 -21093.219} C_VEL
LIN {X 0,Y 153.697,Z 684.691,A -85,B 0,C 180,E1 -21098.675,E2 -21098.675} C_VEL
LIN {X 0,Y 160.141,Z 667.742,A -85,B 0,C 180,E1 -21103.379,E2 -21103.379} C_VEL
LIN {X 0,Y 166.838,Z 649.18,A -85,B 0,C 180,E1 -21107.37,E2 -21107.37} C_VEL
LIN {X 0,Y 173.319,Z 629.638,A -85,B 0,C 180,E1 -21110.629,E2 -21110.629} C_VEL
LIN {X 0,Y 179.516,Z 608.54,A -85,B 0,C 180,E1 -21113.328,E2 -21113.328} C_VEL
LIN {X 0,Y 184.868,Z 587.205,A -85,B 0,C 180,E1 -21115.393,E2 -21115.393} C_VEL
LIN {X 0,Y 189.519,Z 564.35,A -85,B 0,C 180,E1 -21116.987,E2 -21116.987} C_VEL
LIN {X 0,Y 200.571,Z 495.538,A -85,B 0,C 180,E1 -21120.507,E2 -21120.507} C_VEL
LIN {X 0,Y 196.571,Z 500.049,A -85,B 0,C 180,E1 -21121.108,E2 -21121.108} C_VEL
LIN {X 0,Y 192.978,Z 508.1,A -85,B 0,C 180,E1 -21121.287,E2 -21121.287} C_VEL
LIN {X 0,Y 189.976,Z 512.133,A -85,B 0,C 180,E1 -21121.681,E2 -21121.681} C_VEL
LIN {X 0,Y 187.942,Z 514.262,A -85,B 0,C 180,E1 -21122.168,E2 -21122.168} C_VEL
LIN {X 0,Y 187.389,Z 518.122,A -85,B 0,C 180,E1 -21122.596,E2 -21122.596} C_VEL
LIN {X 0,Y 186.904,Z 526.413,A -85,B 0,C 180,E1 -21122.95,E2 -21122.95} C_VEL
LIN {X 0,Y 178.232,Z 635.184,A -85,B 0,C 180,E1 -21126.7,E2 -21126.7} C_VEL
LIN {X 0,Y 175.765,Z 651.989,A -85,B 0,C 180,E1 -21127.835,E2 -21127.835} C_VEL
LIN {X 0,Y 172.642,Z 666.742,A -85,B 0,C 180,E1 -21129.308,E2 -21129.308} C_VEL
LIN {X 0,Y 168.594,Z 681.234,A -85,B 0,C 180,E1 -21131.318,E2 -21131.318} C_VEL
LIN {X 0,Y 163.629,Z 695.775,A -85,B 0,C 180,E1 -21134.036,E2 -21134.036} C_VEL
LIN {X 0,Y 158.471,Z 708.511,A -85,B 0,C 180,E1 -21137.238,E2 -21137.238} C_VEL
LIN {X 0,Y 153.349,Z 719.856,A -85,B 0,C 180,E1 -21140.993,E2 -21140.993} C_VEL
LIN {X 0,Y 148.442,Z 729.85,A -85,B 0,C 180,E1 -21145.36,E2 -21145.36} C_VEL
LIN {X 0,Y 143.727,Z 739.095,A -85,B 0,C 180,E1 -21150.793,E2 -21150.793} C_VEL
LIN {X 0,Y 140.182,Z 746.209,A -85,B 0,C 180,E1 -21156.548,E2 -21156.548} C_VEL
LIN {X 0,Y 137.716,Z 751.82,A -85,B 0,C 180,E1 -21163.002,E2 -21163.002} C_VEL
LIN {X 0,Y 136.594,Z 755.376,A -85,B 0,C 180,E1 -21169.227,E2 -21169.227} C_VEL
LIN {X 0,Y 136.355,Z 757.366,A -85,B 0,C 180,E1 -21175.629,E2 -21175.629} C_VEL
LIN {X 0,Y 136.925,Z 757.835,A -85,B 0,C 180,E1 -21182.207,E2 -21182.207} C_VEL
LIN {X 0,Y 138.691,Z 756.654,A -85,B 0,C 180,E1 -21188.865,E2 -21188.865} C_VEL
LIN {X 0,Y 142.253,Z 753.429,A -85,B 0,C 180,E1 -21195.795,E2 -21195.795} C_VEL
LIN {X 0,Y 147.052,Z 748.647,A -85,B 0,C 180,E1 -21201.774,E2 -21201.774} C_VEL
LIN {X 0,Y 153.218,Z 741.888,A -85,B 0,C 180,E1 -21207.324,E2 -21207.324} C_VEL
LIN {X 0,Y 160.059,Z 733.612,A -85,B 0,C 180,E1 -21212.061,E2 -21212.061} C_VEL
LIN {X 0,Y 167.558,Z 723.336,A -85,B 0,C 180,E1 -21216.253,E2 -21216.253} C_VEL
LIN {X 0,Y 174.867,Z 711.855,A -85,B 0,C 180,E1 -21219.66,E2 -21219.66} C_VEL
LIN {X 0,Y 181.888,Z 698.953,A -85,B 0,C 180,E1 -21222.491,E2 -21222.491} C_VEL
LIN {X 0,Y 188.022,Z 685.345,A -85,B 0,C 180,E1 -21224.695,E2 -21224.695} C_VEL
LIN {X 0,Y 193.337,Z 670.636,A -85,B 0,C 180,E1 -21226.455,E2 -21226.455} C_VEL
LIN {X 0,Y 197.488,Z 655.424,A -85,B 0,C 180,E1 -21227.77,E2 -21227.77} C_VEL
LIN {X 0,Y 200.617,Z 638.602,A -85,B 0,C 180,E1 -21228.754,E2 -21228.754} C_VEL
LIN {X 0,Y 204.02,Z 605.1,A -85,B 0,C 180,E1 -21229.848,E2 -21229.848} C_VEL
LIN {X 0,Y 211.834,Z 524.075,A -85,B 0,C 180,E1 -21232.221,E2 -21232.221} C_VEL
LIN {X 0,Y 212.398,Z 496.448,A -85,B 0,C 180,E1 -21234.427,E2 -21234.427} C_VEL
LIN {X 0,Y 212.772,Z 490.461,A -85,B 0,C 180,E1 -21234.98,E2 -21234.98} C_VEL
LIN {X 0,Y 224.955,Z 447.879,A -85,B 0,C 180,E1 -21240.11,E2 -21240.11} C_VEL
LIN {X 0,Y 225.289,Z 446.689,A -85,B 0,C 180,E1 -21240.253,E2 -21240.253} C_VEL
LIN {X 0,Y 224.925,Z 439.714,A -85,B 0,C 180,E1 -21243.567,E2 -21243.567} C_VEL
LIN {X 0,Y 224.669,Z 434.477,A -85,B 0,C 180,E1 -21247.083,E2 -21247.083} C_VEL
LIN {X 0,Y 224.564,Z 431.171,A -85,B 0,C 180,E1 -21250.286,E2 -21250.286} C_VEL
LIN {X 0,Y 225.058,Z 428.722,A -85,B 0,C 180,E1 -21254.142,E2 -21254.142} C_VEL
LIN {X 0,Y 225.213,Z 428.615,A -85,B 0,C 180,E1 -21255.976,E2 -21255.976} C_VEL
LIN {X 0,Y 223.089,Z 438.023,A -85,B 0,C 180,E1 -21259.497,E2 -21259.497} C_VEL
LIN {X 0,Y 222.438,Z 440.67,A -85,B 0,C 180,E1 -21260.062,E2 -21260.062} C_VEL
LIN {X 0,Y 221.128,Z 444.689,A -85,B 0,C 180,E1 -21260.341,E2 -21260.341} C_VEL
LIN {X 0,Y 216.142,Z 458.259,A -85,B 0,C 180,E1 -21260.192,E2 -21260.192} C_VEL
LIN {X 0,Y 215.382,Z 460.548,A -85,B 0,C 180,E1 -21260.29,E2 -21260.29} C_VEL
LIN {X 0,Y 204.017,Z 497.28,A -85,B 0,C 180,E1 -21262.6,E2 -21262.6} C_VEL
LIN {X 0,Y 194.372,Z 587.356,A -85,B 0,C 180,E1 -21265.803,E2 -21265.803} C_VEL
LIN {X 0,Y 190.852,Z 624.419,A -85,B 0,C 180,E1 -21267.402,E2 -21267.402} C_VEL
LIN {X 0,Y 188.404,Z 647.642,A -85,B 0,C 180,E1 -21268.551,E2 -21268.551} C_VEL
LIN {X 0,Y 185.307,Z 663.835,A -85,B 0,C 180,E1 -21269.761,E2 -21269.761} C_VEL
LIN {X 0,Y 180.934,Z 679.336,A -85,B 0,C 180,E1 -21271.383,E2 -21271.383} C_VEL
LIN {X 0,Y 175.515,Z 694.069,A -85,B 0,C 180,E1 -21273.437,E2 -21273.437} C_VEL
LIN {X 0,Y 169.269,Z 707.769,A -85,B 0,C 180,E1 -21275.985,E2 -21275.985} C_VEL
LIN {X 0,Y 161.79,Z 721.666,A -85,B 0,C 180,E1 -21279.428,E2 -21279.428} C_VEL
LIN {X 0,Y 154.309,Z 733.62,A -85,B 0,C 180,E1 -21283.478,E2 -21283.478} C_VEL
LIN {X 0,Y 147.122,Z 744.014,A -85,B 0,C 180,E1 -21288.246,E2 -21288.246} C_VEL
LIN {X 0,Y 140.559,Z 752.753,A -85,B 0,C 180,E1 -21293.819,E2 -21293.819} C_VEL
LIN {X 0,Y 135.035,Z 759.962,A -85,B 0,C 180,E1 -21300.264,E2 -21300.264} C_VEL
LIN {X 0,Y 131.03,Z 765.309,A -85,B 0,C 180,E1 -21307.414,E2 -21307.414} C_VEL
LIN {X 0,Y 128.834,Z 768.723,A -85,B 0,C 180,E1 -21314.706,E2 -21314.706} C_VEL
LIN {X 0,Y 128.211,Z 770.292,A -85,B 0,C 180,E1 -21322.049,E2 -21322.049} C_VEL
LIN {X 0,Y 128.388,Z 770.241,A -85,B 0,C 180,E1 -21328.22,E2 -21328.22} C_VEL
LIN {X 0,Y 128.386,Z 769.096,A -85,B 0,C 180,E1 -21333.577,E2 -21333.577} C_VEL
LIN {X 0,Y 128.497,Z 766.359,A -85,B 0,C 180,E1 -21339.862,E2 -21339.862} C_VEL
LIN {X 0,Y 128.816,Z 764.854,A -85,B 0,C 180,E1 -21342.557,E2 -21342.557} C_VEL
LIN {X 0,Y 131.253,Z 766.254,A -85,B 0,C 180,E1 -21352.866,E2 -21352.866} C_VEL
LIN {X 0,Y 138.611,Z 765.981,A -85,B 0,C 180,E1 -21363.745,E2 -21363.745} C_VEL
LIN {X 0,Y 152.308,Z 763.787,A -85,B 0,C 180,E1 -21374.101,E2 -21374.101} C_VEL
LIN {X 0,Y 160.499,Z 762.17,A -85,B 0,C 180,E1 -21378.289,E2 -21378.289} C_VEL
LIN {X 0,Y 146.19,Z 761.822,A -85,B 0,C 180,E1 -21386.36,E2 -21386.36} C_VEL
LIN {X 0,Y 136.487,Z 759.886,A -85,B 0,C 180,E1 -21395.321,E2 -21395.321} C_VEL
LIN {X 0,Y 130.847,Z 756.352,A -85,B 0,C 180,E1 -21404.943,E2 -21404.943} C_VEL
LIN {X 0,Y 128.672,Z 751.44,A -85,B 0,C 180,E1 -21414.204,E2 -21414.204} C_VEL
LIN {X 0,Y 128.309,Z 746.391,A -85,B 0,C 180,E1 -21421.341,E2 -21421.341} C_VEL
LIN {X 0,Y 128.557,Z 739.855,A -85,B 0,C 180,E1 -21428.5,E2 -21428.5} C_VEL
LIN {X 0,Y 129.878,Z 731.149,A -85,B 0,C 180,E1 -21436.092,E2 -21436.092} C_VEL
LIN {X 0,Y 132.724,Z 720.359,A -85,B 0,C 180,E1 -21443.534,E2 -21443.534} C_VEL
LIN {X 0,Y 136.933,Z 708.027,A -85,B 0,C 180,E1 -21450.255,E2 -21450.255} C_VEL
LIN {X 0,Y 142.425,Z 693.704,A -85,B 0,C 180,E1 -21456.387,E2 -21456.387} C_VEL
LIN {X 0,Y 148.518,Z 678.345,A -85,B 0,C 180,E1 -21461.541,E2 -21461.541} C_VEL
LIN {X 0,Y 155.327,Z 660.805,A -85,B 0,C 180,E1 -21466.136,E2 -21466.136} C_VEL
LIN {X 0,Y 162.096,Z 642.235,A -85,B 0,C 180,E1 -21469.898,E2 -21469.898} C_VEL
LIN {X 0,Y 168.842,Z 621.674,A -85,B 0,C 180,E1 -21473.08,E2 -21473.08} C_VEL
LIN {X 0,Y 175.053,Z 600.001,A -85,B 0,C 180,E1 -21475.626,E2 -21475.626} C_VEL
LIN {X 0,Y 180.378,Z 577.861,A -85,B 0,C 180,E1 -21477.561,E2 -21477.561} C_VEL
LIN {X 0,Y 184.939,Z 553.575,A -85,B 0,C 180,E1 -21479.05,E2 -21479.05} C_VEL
LIN {X 0,Y 189.625,Z 524.883,A -85,B 0,C 180,E1 -21480.578,E2 -21480.578} C_VEL
LIN {X 0,Y 185.421,Z 534.382,A -85,B 0,C 180,E1 -21480.745,E2 -21480.745} C_VEL
LIN {X 0,Y 182.143,Z 538.992,A -85,B 0,C 180,E1 -21481.155,E2 -21481.155} C_VEL
LIN {X 0,Y 180.549,Z 542.085,A -85,B 0,C 180,E1 -21481.53,E2 -21481.53} C_VEL
LIN {X 0,Y 179.354,Z 551.32,A -85,B 0,C 180,E1 -21481.955,E2 -21481.955} C_VEL
LIN {X 0,Y 172.354,Z 635.636,A -85,B 0,C 180,E1 -21484.93,E2 -21484.93} C_VEL
LIN {X 0,Y 169.761,Z 652.518,A -85,B 0,C 180,E1 -21486.087,E2 -21486.087} C_VEL
LIN {X 0,Y 166.535,Z 667.111,A -85,B 0,C 180,E1 -21487.567,E2 -21487.567} C_VEL
LIN {X 0,Y 162.279,Z 681.697,A -85,B 0,C 180,E1 -21489.624,E2 -21489.624} C_VEL
LIN {X 0,Y 157.086,Z 696.228,A -85,B 0,C 180,E1 -21492.398,E2 -21492.398} C_VEL
LIN {X 0,Y 151.421,Z 709.519,A -85,B 0,C 180,E1 -21495.854,E2 -21495.854} C_VEL
LIN {X 0,Y 146.063,Z 720.768,A -85,B 0,C 180,E1 -21499.744,E2 -21499.744} C_VEL
LIN {X 0,Y 140.524,Z 731.368,A -85,B 0,C 180,E1 -21504.688,E2 -21504.688} C_VEL
LIN {X 0,Y 135.971,Z 739.819,A -85,B 0,C 180,E1 -21509.995,E2 -21509.995} C_VEL
LIN {X 0,Y 132.256,Z 746.841,A -85,B 0,C 180,E1 -21516.071,E2 -21516.071} C_VEL
LIN {X 0,Y 129.696,Z 752.395,A -85,B 0,C 180,E1 -21522.914,E2 -21522.914} C_VEL
LIN {X 0,Y 128.544,Z 755.948,A -85,B 0,C 180,E1 -21529.744,E2 -21529.744} C_VEL
LIN {X 0,Y 128.396,Z 757.896,A -85,B 0,C 180,E1 -21536.845,E2 -21536.845} C_VEL
LIN {X 0,Y 129.213,Z 758.215,A -85,B 0,C 180,E1 -21543.852,E2 -21543.852} C_VEL
LIN {X 0,Y 131.554,Z 756.704,A -85,B 0,C 180,E1 -21551.196,E2 -21551.196} C_VEL
LIN {X 0,Y 135.603,Z 753.414,A -85,B 0,C 180,E1 -21558.127,E2 -21558.127} C_VEL
LIN {X 0,Y 141.262,Z 748.146,A -85,B 0,C 180,E1 -21564.519,E2 -21564.519} C_VEL
LIN {X 0,Y 147.897,Z 741.367,A -85,B 0,C 180,E1 -21569.98,E2 -21569.98} C_VEL
LIN {X 0,Y 155.646,Z 732.426,A -85,B 0,C 180,E1 -21574.916,E2 -21574.916} C_VEL
LIN {X 0,Y 163.193,Z 722.607,A -85,B 0,C 180,E1 -21578.807,E2 -21578.807} C_VEL
LIN {X 0,Y 170.7,Z 711.251,A -85,B 0,C 180,E1 -21582.074,E2 -21582.074} C_VEL
LIN {X 0,Y 177.733,Z 698.817,A -85,B 0,C 180,E1 -21584.735,E2 -21584.735} C_VEL
LIN {X 0,Y 184.25,Z 684.766,A -85,B 0,C 180,E1 -21586.94,E2 -21586.94} C_VEL
LIN {X 0,Y 189.682,Z 670.139,A -85,B 0,C 180,E1 -21588.632,E2 -21588.632} C_VEL
LIN {X 0,Y 194.005,Z 654.43,A -85,B 0,C 180,E1 -21589.927,E2 -21589.927} C_VEL
LIN {X 0,Y 197.094,Z 637.969,A -85,B 0,C 180,E1 -21590.846,E2 -21590.846} C_VEL
LIN {X 0,Y 208.623,Z 525.21,A -85,B 0,C 180,E1 -21594.204,E2 -21594.204} C_VEL
LIN {X 0,Y 209.509,Z 497.097,A -85,B 0,C 180,E1 -21596.493,E2 -21596.493} C_VEL
LIN {X 0,Y 209.986,Z 490.835,A -85,B 0,C 180,E1 -21597.087,E2 -21597.087} C_VEL
LIN {X 0,Y 221.687,Z 451.523,A -85,B 0,C 180,E1 -21601.776,E2 -21601.776} C_VEL
LIN {X 0,Y 221.644,Z 445.832,A -85,B 0,C 180,E1 -21604.657,E2 -21604.657} C_VEL
LIN {X 0,Y 221.626,Z 441.035,A -85,B 0,C 180,E1 -21608.039,E2 -21608.039} C_VEL
LIN {X 0,Y 221.723,Z 438.353,A -85,B 0,C 180,E1 -21610.917,E2 -21610.917} C_VEL
LIN {X 0,Y 222.268,Z 436.205,A -85,B 0,C 180,E1 -21614.324,E2 -21614.324} C_VEL
LIN {X 0,Y 222.344,Z 436.178,A -85,B 0,C 180,E1 -21615.385,E2 -21615.385} C_VEL
LIN {X 0,Y 219.694,Z 447.341,A -85,B 0,C 180,E1 -21619.509,E2 -21619.509} C_VEL
LIN {X 0,Y 215.382,Z 460.548,A -85,B 0,C 180,E1 -21620.29,E2 -21620.29} C_VEL
LIN {X 0,Y 212.886,Z 467.853,A -85,B 0,C 180,E1 -21620.486,E2 -21620.486} C_VEL
LIN {X 0,Y 205.414,Z 487.683,A -85,B 0,C 180,E1 -21619.979,E2 -21619.979} C_VEL
LIN {X 0,Y 203.249,Z 493.872,A -85,B 0,C 180,E1 -21620.186,E2 -21620.186} C_VEL
LIN {X 0,Y 202.069,Z 500.702,A -85,B 0,C 180,E1 -21620.5,E2 -21620.5} C_VEL
LIN {X 0,Y 192.265,Z 588.417,A -85,B 0,C 180,E1 -21623.533,E2 -21623.533} C_VEL
LIN {X 0,Y 188.432,Z 625.593,A -85,B 0,C 180,E1 -21625.125,E2 -21625.125} C_VEL
LIN {X 0,Y 185.928,Z 647.063,A -85,B 0,C 180,E1 -21626.174,E2 -21626.174} C_VEL
LIN {X 0,Y 182.619,Z 663.38,A -85,B 0,C 180,E1 -21627.344,E2 -21627.344} C_VEL
LIN {X 0,Y 178.11,Z 678.587,A -85,B 0,C 180,E1 -21628.876,E2 -21628.876} C_VEL
LIN {X 0,Y 172.036,Z 694.227,A -85,B 0,C 180,E1 -21630.998,E2 -21630.998} C_VEL
LIN {X 0,Y 165.087,Z 708.426,A -85,B 0,C 180,E1 -21633.623,E2 -21633.623} C_VEL
LIN {X 0,Y 157.471,Z 721.539,A -85,B 0,C 180,E1 -21636.874,E2 -21636.874} C_VEL
LIN {X 0,Y 149.139,Z 733.82,A -85,B 0,C 180,E1 -21641.071,E2 -21641.071} C_VEL
LIN {X 0,Y 141.683,Z 743.714,A -85,B 0,C 180,E1 -21645.689,E2 -21645.689} C_VEL
LIN {X 0,Y 134.485,Z 752.399,A -85,B 0,C 180,E1 -21651.36,E2 -21651.36} C_VEL
LIN {X 0,Y 128.322,Z 759.579,A -85,B 0,C 180,E1 -21658.011,E2 -21658.011} C_VEL
LIN {X 0,Y 123.87,Z 764.727,A -85,B 0,C 180,E1 -21665.188,E2 -21665.188} C_VEL
LIN {X 0,Y 121.103,Z 768.31,A -85,B 0,C 180,E1 -21673.209,E2 -21673.209} C_VEL
LIN {X 0,Y 120.228,Z 769.872,A -85,B 0,C 180,E1 -21680.914,E2 -21680.914} C_VEL
LIN {X 0,Y 120.376,Z 769.844,A -85,B 0,C 180,E1 -21687.625,E2 -21687.625} C_VEL
LIN {X 0,Y 120.409,Z 768.863,A -85,B 0,C 180,E1 -21692.861,E2 -21692.861} C_VEL
LIN {X 0,Y 120.475,Z 766.241,A -85,B 0,C 180,E1 -21699.56,E2 -21699.56} C_VEL
LIN {X 0,Y 121.104,Z 763.691,A -85,B 0,C 180,E1 -21704.346,E2 -21704.346} C_VEL
LIN {X 0,Y 124.727,Z 765.297,A -85,B 0,C 180,E1 -21716.167,E2 -21716.167} C_VEL
LIN {X 0,Y 134.486,Z 765.11,A -85,B 0,C 180,E1 -21728.108,E2 -21728.108} C_VEL
LIN {X 0,Y 149.618,Z 763.223,A -85,B 0,C 180,E1 -21737.889,E2 -21737.889} C_VEL
LIN {X 0,Y 150.332,Z 763.087,A -85,B 0,C 180,E1 -21738.312,E2 -21738.312} C_VEL
LIN {X 0,Y 136.634,Z 761.817,A -85,B 0,C 180,E1 -21746.715,E2 -21746.715} C_VEL
LIN {X 0,Y 126.957,Z 758.851,A -85,B 0,C 180,E1 -21756.812,E2 -21756.812} C_VEL
LIN {X 0,Y 122.02,Z 754.358,A -85,B 0,C 180,E1 -21767.22,E2 -21767.22} C_VEL
LIN {X 0,Y 120.548,Z 749.125,A -85,B 0,C 180,E1 -21776.197,E2 -21776.197} C_VEL
LIN {X 0,Y 120.361,Z 743.74,A -85,B 0,C 180,E1 -21783.335,E2 -21783.335} C_VEL
LIN {X 0,Y 120.871,Z 736.504,A -85,B 0,C 180,E1 -21790.97,E2 -21790.97} C_VEL
LIN {X 0,Y 122.746,Z 726.938,A -85,B 0,C 180,E1 -21799.018,E2 -21799.018} C_VEL
LIN {X 0,Y 126.078,Z 715.923,A -85,B 0,C 180,E1 -21806.368,E2 -21806.368} C_VEL
LIN {X 0,Y 130.65,Z 703.573,A -85,B 0,C 180,E1 -21812.915,E2 -21812.915} C_VEL
LIN {X 0,Y 136.581,Z 688.898,A -85,B 0,C 180,E1 -21819.021,E2 -21819.021} C_VEL
LIN {X 0,Y 143.505,Z 671.986,A -85,B 0,C 180,E1 -21824.447,E2 -21824.447} C_VEL
LIN {X 0,Y 150.649,Z 653.881,A -85,B 0,C 180,E1 -21828.919,E2 -21828.919} C_VEL
LIN {X 0,Y 157.86,Z 634.093,A -85,B 0,C 180,E1 -21832.648,E2 -21832.648} C_VEL
LIN {X 0,Y 164.696,Z 612.92,A -85,B 0,C 180,E1 -21835.657,E2 -21835.657} C_VEL
LIN {X 0,Y 170.893,Z 590.458,A -85,B 0,C 180,E1 -21838.037,E2 -21838.037} C_VEL
LIN {X 0,Y 176.11,Z 567.409,A -85,B 0,C 180,E1 -21839.802,E2 -21839.802} C_VEL
LIN {X 0,Y 176.372,Z 565.823,A -85,B 0,C 180,E1 -21839.909,E2 -21839.909} C_VEL
LIN {X 0,Y 173.022,Z 569.857,A -85,B 0,C 180,E1 -21840.482,E2 -21840.482} C_VEL
LIN {X 0,Y 171.941,Z 575.213,A -85,B 0,C 180,E1 -21840.828,E2 -21840.828} C_VEL
LIN {X 0,Y 166.523,Z 636.559,A -85,B 0,C 180,E1 -21843.087,E2 -21843.087} C_VEL
LIN {X 0,Y 163.719,Z 653.78,A -85,B 0,C 180,E1 -21844.299,E2 -21844.299} C_VEL
LIN {X 0,Y 160.202,Z 668.669,A -85,B 0,C 180,E1 -21845.867,E2 -21845.867} C_VEL
LIN {X 0,Y 155.492,Z 683.807,A -85,B 0,C 180,E1 -21848.098,E2 -21848.098} C_VEL
LIN {X 0,Y 150.342,Z 697.358,A -85,B 0,C 180,E1 -21850.805,E2 -21850.805} C_VEL
LIN {X 0,Y 144.245,Z 710.887,A -85,B 0,C 180,E1 -21854.478,E2 -21854.478} C_VEL
LIN {X 0,Y 138.832,Z 721.611,A -85,B 0,C 180,E1 -21858.376,E2 -21858.376} C_VEL
LIN {X 0,Y 133.031,Z 732.092,A -85,B 0,C 180,E1 -21863.522,E2 -21863.522} C_VEL
LIN {X 0,Y 128.241,Z 740.48,A -85,B 0,C 180,E1 -21869.102,E2 -21869.102} C_VEL
LIN {X 0,Y 124.337,Z 747.428,A -85,B 0,C 180,E1 -21875.532,E2 -21875.532} C_VEL
LIN {X 0,Y 121.672,Z 752.937,A -85,B 0,C 180,E1 -21882.814,E2 -21882.814} C_VEL
LIN {X 0,Y 120.494,Z 756.527,A -85,B 0,C 180,E1 -21890.391,E2 -21890.391} C_VEL
LIN {X 0,Y 120.441,Z 758.339,A -85,B 0,C 180,E1 -21897.697,E2 -21897.697} C_VEL
LIN {X 0,Y 121.474,Z 758.594,A -85,B 0,C 180,E1 -21905.175,E2 -21905.175} C_VEL
LIN {X 0,Y 124.311,Z 756.97,A -85,B 0,C 180,E1 -21913.124,E2 -21913.124} C_VEL
LIN {X 0,Y 128.808,Z 753.656,A -85,B 0,C 180,E1 -21920.209,E2 -21920.209} C_VEL
LIN {X 0,Y 135.028,Z 748.367,A -85,B 0,C 180,E1 -21926.788,E2 -21926.788} C_VEL
LIN {X 0,Y 142.225,Z 741.57,A -85,B 0,C 180,E1 -21932.354,E2 -21932.354} C_VEL
LIN {X 0,Y 149.895,Z 733.32,A -85,B 0,C 180,E1 -21936.989,E2 -21936.989} C_VEL
LIN {X 0,Y 158.003,Z 723.418,A -85,B 0,C 180,E1 -21940.975,E2 -21940.975} C_VEL
LIN {X 0,Y 165.979,Z 712.006,A -85,B 0,C 180,E1 -21944.27,E2 -21944.27} C_VEL
LIN {X 0,Y 173.692,Z 698.979,A -85,B 0,C 180,E1 -21947.025,E2 -21947.025} C_VEL
LIN {X 0,Y 180.303,Z 685.284,A -85,B 0,C 180,E1 -21949.131,E2 -21949.131} C_VEL
LIN {X 0,Y 186.029,Z 670.575,A -85,B 0,C 180,E1 -21950.805,E2 -21950.805} C_VEL
LIN {X 0,Y 190.559,Z 654.847,A -85,B 0,C 180,E1 -21952.079,E2 -21952.079} C_VEL
LIN {X 0,Y 193.788,Z 638.43,A -85,B 0,C 180,E1 -21952.978,E2 -21952.978} C_VEL
LIN {X 0,Y 204.209,Z 541.284,A -85,B 0,C 180,E1 -21955.789,E2 -21955.789} C_VEL
LIN {X 0,Y 205.73,Z 526.209,A -85,B 0,C 180,E1 -21956.261,E2 -21956.261} C_VEL
LIN {X 0,Y 206.965,Z 497.506,A -85,B 0,C 180,E1 -21958.643,E2 -21958.643} C_VEL
LIN {X 0,Y 207.351,Z 491.943,A -85,B 0,C 180,E1 -21959.17,E2 -21959.17} C_VEL
LIN {X 0,Y 218.321,Z 456.356,A -85,B 0,C 180,E1 -21963.379,E2 -21963.379} C_VEL
LIN {X 0,Y 218.508,Z 451.219,A -85,B 0,C 180,E1 -21966.304,E2 -21966.304} C_VEL
LIN {X 0,Y 218.611,Z 447.258,A -85,B 0,C 180,E1 -21969.476,E2 -21969.476} C_VEL
LIN {X 0,Y 218.922,Z 445.339,A -85,B 0,C 180,E1 -21971.859,E2 -21971.859} C_VEL
LIN {X 0,Y 219.533,Z 443.702,A -85,B 0,C 180,E1 -21974.742,E2 -21974.742} C_VEL
LIN {X 0,Y 217.397,Z 451.382,A -85,B 0,C 180,E1 -21977.612,E2 -21977.612} C_VEL
LIN {X 0,Y 203.249,Z 493.872,A -85,B 0,C 180,E1 -21980.186,E2 -21980.186} C_VEL
LIN {X 0,Y 202.26,Z 498.075,A -85,B 0,C 180,E1 -21980.24,E2 -21980.24} C_VEL
LIN {X 0,Y 198.78,Z 519.875,A -85,B 0,C 180,E1 -21979.13,E2 -21979.13} C_VEL
LIN {X 0,Y 197.506,Z 528.802,A -85,B 0,C 180,E1 -21979.132,E2 -21979.132} C_VEL
LIN {X 0,Y 190.628,Z 588.136,A -85,B 0,C 180,E1 -21981.174,E2 -21981.174} C_VEL
LIN {X 0,Y 186.453,Z 626.377,A -85,B 0,C 180,E1 -21982.763,E2 -21982.763} C_VEL
LIN {X 0,Y 183.974,Z 646.407,A -85,B 0,C 180,E1 -21983.725,E2 -21983.725} C_VEL
LIN {X 0,Y 180.416,Z 662.83,A -85,B 0,C 180,E1 -21984.849,E2 -21984.849} C_VEL
LIN {X 0,Y 175.31,Z 678.869,A -85,B 0,C 180,E1 -21986.413,E2 -21986.413} C_VEL
LIN {X 0,Y 168.886,Z 694.356,A -85,B 0,C 180,E1 -21988.467,E2 -21988.467} C_VEL
LIN {X 0,Y 161.203,Z 709.08,A -85,B 0,C 180,E1 -21991.145,E2 -21991.145} C_VEL
LIN {X 0,Y 153.5,Z 721.472,A -85,B 0,C 180,E1 -21994.192,E2 -21994.192} C_VEL
LIN {X 0,Y 144.943,Z 733.227,A -85,B 0,C 180,E1 -21998.157,E2 -21998.157} C_VEL
LIN {X 0,Y 136.559,Z 743.443,A -85,B 0,C 180,E1 -22002.938,E2 -22002.938} C_VEL
LIN {X 0,Y 128.697,Z 752.084,A -85,B 0,C 180,E1 -22008.679,E2 -22008.679} C_VEL
LIN {X 0,Y 121.835,Z 759.211,A -85,B 0,C 180,E1 -22015.517,E2 -22015.517} C_VEL
LIN {X 0,Y 116.493,Z 764.602,A -85,B 0,C 180,E1 -22023.499,E2 -22023.499} C_VEL
LIN {X 0,Y 113.45,Z 767.902,A -85,B 0,C 180,E1 -22031.508,E2 -22031.508} C_VEL
LIN {X 0,Y 112.268,Z 769.46,A -85,B 0,C 180,E1 -22039.745,E2 -22039.745} C_VEL
LIN {X 0,Y 112.358,Z 769.441,A -85,B 0,C 180,E1 -22046.945,E2 -22046.945} C_VEL
LIN {X 0,Y 112.427,Z 768.471,A -85,B 0,C 180,E1 -22052.554,E2 -22052.554} C_VEL
LIN {X 0,Y 112.49,Z 765.856,A -85,B 0,C 180,E1 -22059.728,E2 -22059.728} C_VEL
LIN {X 0,Y 113.523,Z 762.407,A -85,B 0,C 180,E1 -22066.376,E2 -22066.376} C_VEL
LIN {X 0,Y 118.347,Z 764.275,A -85,B 0,C 180,E1 -22079.347,E2 -22079.347} C_VEL
LIN {X 0,Y 129.663,Z 764.361,A -85,B 0,C 180,E1 -22091.547,E2 -22091.547} C_VEL
LIN {X 0,Y 140.208,Z 763.444,A -85,B 0,C 180,E1 -22098.32,E2 -22098.32} C_VEL
LIN {X 0,Y 126.639,Z 761.21,A -85,B 0,C 180,E1 -22107.53,E2 -22107.53} C_VEL
LIN {X 0,Y 117.821,Z 757.452,A -85,B 0,C 180,E1 -22118.077,E2 -22118.077} C_VEL
LIN {X 0,Y 113.602,Z 752.346,A -85,B 0,C 180,E1 -22128.837,E2 -22128.837} C_VEL
LIN {X 0,Y 112.526,Z 746.75,A -85,B 0,C 180,E1 -22137.965,E2 -22137.965} C_VEL
LIN {X 0,Y 112.485,Z 740.692,A -85,B 0,C 180,E1 -22145.613,E2 -22145.613} C_VEL
LIN {X 0,Y 113.448,Z 732.262,A -85,B 0,C 180,E1 -22154.174,E2 -22154.174} C_VEL
LIN {X 0,Y 115.92,Z 722.215,A -85,B 0,C 180,E1 -22162.306,E2 -22162.306} C_VEL
LIN {X 0,Y 120.065,Z 710.209,A -85,B 0,C 180,E1 -22169.986,E2 -22169.986} C_VEL
LIN {X 0,Y 125.684,Z 696.284,A -85,B 0,C 180,E1 -22176.917,E2 -22176.917} C_VEL
LIN {X 0,Y 132.27,Z 680.786,A -85,B 0,C 180,E1 -22182.872,E2 -22182.872} C_VEL
LIN {X 0,Y 139.729,Z 663.027,A -85,B 0,C 180,E1 -22188.092,E2 -22188.092} C_VEL
LIN {X 0,Y 147.2,Z 644.11,A -85,B 0,C 180,E1 -22192.31,E2 -22192.31} C_VEL
LIN {X 0,Y 154.363,Z 624.096,A -85,B 0,C 180,E1 -22195.695,E2 -22195.695} C_VEL
LIN {X 0,Y 161.807,Z 603.088,A -85,B 0,C 180,E1 -22198.727,E2 -22198.727} C_VEL
LIN {X 0,Y 164.493,Z 598.733,A -85,B 0,C 180,E1 -22199.62,E2 -22199.62} C_VEL
LIN {X 0,Y 160.873,Z 637.386,A -85,B 0,C 180,E1 -22201.112,E2 -22201.112} C_VEL
LIN {X 0,Y 157.89,Z 654.784,A -85,B 0,C 180,E1 -22202.359,E2 -22202.359} C_VEL
LIN {X 0,Y 154.053,Z 670.031,A -85,B 0,C 180,E1 -22204.013,E2 -22204.013} C_VEL
LIN {X 0,Y 149.146,Z 684.985,A -85,B 0,C 180,E1 -22206.278,E2 -22206.278} C_VEL
LIN {X 0,Y 143.783,Z 698.304,A -85,B 0,C 180,E1 -22209.03,E2 -22209.03} C_VEL
LIN {X 0,Y 137.405,Z 711.746,A -85,B 0,C 180,E1 -22212.801,E2 -22212.801} C_VEL
LIN {X 0,Y 131.214,Z 723.232,A -85,B 0,C 180,E1 -22217.229,E2 -22217.229} C_VEL
LIN {X 0,Y 125.17,Z 733.536,A -85,B 0,C 180,E1 -22222.652,E2 -22222.652} C_VEL
LIN {X 0,Y 120.012,Z 741.969,A -85,B 0,C 180,E1 -22228.837,E2 -22228.837} C_VEL
LIN {X 0,Y 115.964,Z 748.873,A -85,B 0,C 180,E1 -22235.933,E2 -22235.933} C_VEL
LIN {X 0,Y 113.521,Z 753.745,A -85,B 0,C 180,E1 -22243.232,E2 -22243.232} C_VEL
LIN {X 0,Y 112.436,Z 757.188,A -85,B 0,C 180,E1 -22251.377,E2 -22251.377} C_VEL
LIN {X 0,Y 112.552,Z 758.865,A -85,B 0,C 180,E1 -22259.242,E2 -22259.242} C_VEL
LIN {X 0,Y 113.957,Z 758.904,A -85,B 0,C 180,E1 -22267.251,E2 -22267.251} C_VEL
LIN {X 0,Y 117.476,Z 757.108,A -85,B 0,C 180,E1 -22275.737,E2 -22275.737} C_VEL
LIN {X 0,Y 122.637,Z 753.604,A -85,B 0,C 180,E1 -22283.025,E2 -22283.025} C_VEL
LIN {X 0,Y 129.62,Z 748.167,A -85,B 0,C 180,E1 -22289.751,E2 -22289.751} C_VEL
LIN {X 0,Y 137.503,Z 741.119,A -85,B 0,C 180,E1 -22295.347,E2 -22295.347} C_VEL
LIN {X 0,Y 145.8,Z 732.663,A -85,B 0,C 180,E1 -22299.955,E2 -22299.955} C_VEL
LIN {X 0,Y 154.332,Z 722.595,A -85,B 0,C 180,E1 -22303.823,E2 -22303.823} C_VEL
LIN {X 0,Y 163.058,Z 710.546,A -85,B 0,C 180,E1 -22307.134,E2 -22307.134} C_VEL
LIN {X 0,Y 170.737,Z 697.845,A -85,B 0,C 180,E1 -22309.658,E2 -22309.658} C_VEL
LIN {X 0,Y 177.81,Z 683.535,A -85,B 0,C 180,E1 -22311.731,E2 -22311.731} C_VEL
LIN {X 0,Y 183.475,Z 668.875,A -85,B 0,C 180,E1 -22313.271,E2 -22313.271} C_VEL
LIN {X 0,Y 188.147,Z 652.528,A -85,B 0,C 180,E1 -22314.491,E2 -22314.491} C_VEL
LIN {X 0,Y 191.134,Z 636.437,A -85,B 0,C 180,E1 -22315.278,E2 -22315.278} C_VEL
LIN {X 0,Y 203.102,Z 527.426,A -85,B 0,C 180,E1 -22318.359,E2 -22318.359} C_VEL
LIN {X 0,Y 204.798,Z 497.863,A -85,B 0,C 180,E1 -22320.856,E2 -22320.856} C_VEL
LIN {X 0,Y 205.236,Z 492.312,A -85,B 0,C 180,E1 -22321.395,E2 -22321.395} C_VEL
LIN {X 0,Y 215.194,Z 461.424,A -85,B 0,C 180,E1 -22324.997,E2 -22324.997} C_VEL
LIN {X 0,Y 215.522,Z 456.686,A -85,B 0,C 180,E1 -22327.999,E2 -22327.999} C_VEL
LIN {X 0,Y 216.015,Z 453.147,A -85,B 0,C 180,E1 -22331.479,E2 -22331.479} C_VEL
LIN {X 0,Y 216.573,Z 451.528,A -85,B 0,C 180,E1 -22334.199,E2 -22334.199} C_VEL
LIN {X 0,Y 215.212,Z 455.651,A -85,B 0,C 180,E1 -22335.701,E2 -22335.701} C_VEL
LIN {X 0,Y 201.415,Z 496.275,A -85,B 0,C 180,E1 -22338.061,E2 -22338.061} C_VEL
LIN {X 0,Y 197.506,Z 528.802,A -85,B 0,C 180,E1 -22339.132,E2 -22339.132} C_VEL
LIN {X 0,Y 196.458,Z 536.499,A -85,B 0,C 180,E1 -22339.086,E2 -22339.086} C_VEL
LIN {X 0,Y 193.171,Z 557.121,A -85,B 0,C 180,E1 -22337.954,E2 -22337.954} C_VEL
LIN {X 0,Y 192.277,Z 563.71,A -85,B 0,C 180,E1 -22337.966,E2 -22337.966} C_VEL
LIN {X 0,Y 188.845,Z 591.771,A -85,B 0,C 180,E1 -22338.899,E2 -22338.899} C_VEL
LIN {X 0,Y 183.238,Z 640.154,A -85,B 0,C 180,E1 -22340.928,E2 -22340.928} C_VEL
LIN {X 0,Y 180.226,Z 656.172,A -85,B 0,C 180,E1 -22341.867,E2 -22341.867} C_VEL
LIN {X 0,Y 176.001,Z 670.839,A -85,B 0,C 180,E1 -22343.038,E2 -22343.038} C_VEL
LIN {X 0,Y 170.343,Z 685.58,A -85,B 0,C 180,E1 -22344.628,E2 -22344.628} C_VEL
LIN {X 0,Y 163.383,Z 699.895,A -85,B 0,C 180,E1 -22346.696,E2 -22346.696} C_VEL
LIN {X 0,Y 154.654,Z 714.434,A -85,B 0,C 180,E1 -22349.602,E2 -22349.602} C_VEL
LIN {X 0,Y 146.309,Z 726.212,A -85,B 0,C 180,E1 -22352.809,E2 -22352.809} C_VEL
LIN {X 0,Y 136.813,Z 737.724,A -85,B 0,C 180,E1 -22357.202,E2 -22357.202} C_VEL
LIN {X 0,Y 128.198,Z 746.932,A -85,B 0,C 180,E1 -22362.197,E2 -22362.197} C_VEL
LIN {X 0,Y 119.51,Z 755.281,A -85,B 0,C 180,E1 -22368.846,E2 -22368.846} C_VEL
LIN {X 0,Y 112.825,Z 761.327,A -85,B 0,C 180,E1 -22376.068,E2 -22376.068} C_VEL
LIN {X 0,Y 107.686,Z 765.854,A -85,B 0,C 180,E1 -22384.723,E2 -22384.723} C_VEL
LIN {X 0,Y 104.977,Z 768.395,A -85,B 0,C 180,E1 -22393.404,E2 -22393.404} C_VEL
LIN {X 0,Y 104.235,Z 769.208,A -85,B 0,C 180,E1 -22402.288,E2 -22402.288} C_VEL
LIN {X 0,Y 104.471,Z 768.618,A -85,B 0,C 180,E1 -22409.458,E2 -22409.458} C_VEL
LIN {X 0,Y 104.396,Z 766.96,A -85,B 0,C 180,E1 -22416.053,E2 -22416.053} C_VEL
LIN {X 0,Y 105.046,Z 763.277,A -85,B 0,C 180,E1 -22424.334,E2 -22424.334} C_VEL
LIN {X 0,Y 106.049,Z 760.985,A -85,B 0,C 180,E1 -22428.418,E2 -22428.418} C_VEL
LIN {X 0,Y 111.495,Z 763.024,A -85,B 0,C 180,E1 -22441.581,E2 -22441.581} C_VEL
LIN {X 0,Y 124.247,Z 763.462,A -85,B 0,C 180,E1 -22454.443,E2 -22454.443} C_VEL
LIN {X 0,Y 130.103,Z 763.244,A -85,B 0,C 180,E1 -22458.338,E2 -22458.338} C_VEL
LIN {X 0,Y 116.705,Z 760.043,A -85,B 0,C 180,E1 -22468.494,E2 -22468.494} C_VEL
LIN {X 0,Y 108.529,Z 755.342,A -85,B 0,C 180,E1 -22480.072,E2 -22480.072} C_VEL
LIN {X 0,Y 105.183,Z 749.524,A -85,B 0,C 180,E1 -22491.379,E2 -22491.379} C_VEL
LIN {X 0,Y 104.542,Z 743.958,A -85,B 0,C 180,E1 -22500.002,E2 -22500.002} C_VEL
LIN {X 0,Y 104.707,Z 737.221,A -85,B 0,C 180,E1 -22508.237,E2 -22508.237} C_VEL
LIN {X 0,Y 106.104,Z 728.423,A -85,B 0,C 180,E1 -22516.987,E2 -22516.987} C_VEL
LIN {X 0,Y 109.224,Z 717.705,A -85,B 0,C 180,E1 -22525.485,E2 -22525.485} C_VEL
LIN {X 0,Y 113.812,Z 705.683,A -85,B 0,C 180,E1 -22533.005,E2 -22533.005} C_VEL
LIN {X 0,Y 120.178,Z 690.866,A -85,B 0,C 180,E1 -22540.152,E2 -22540.152} C_VEL
LIN {X 0,Y 127.482,Z 674.351,A -85,B 0,C 180,E1 -22546.187,E2 -22546.187} C_VEL
LIN {X 0,Y 135.883,Z 655.591,A -85,B 0,C 180,E1 -22551.599,E2 -22551.599} C_VEL
LIN {X 0,Y 137.445,Z 653.713,A -85,B 0,C 180,E1 -22552.463,E2 -22552.463} C_VEL
LIN {X 0,Y 141.396,Z 650.325,A -85,B 0,C 180,E1 -22554.066,E2 -22554.066} C_VEL
LIN {X 0,Y 147.121,Z 643.313,A -85,B 0,C 180,E1 -22555.839,E2 -22555.839} C_VEL
LIN {X 0,Y 153.534,Z 632.723,A -85,B 0,C 180,E1 -22557.584,E2 -22557.584} C_VEL
LIN {X 0,Y 156.742,Z 626.402,A -85,B 0,C 180,E1 -22558.457,E2 -22558.457} C_VEL
LIN {X 0,Y 154.573,Z 643.891,A -85,B 0,C 180,E1 -22559.337,E2 -22559.337} C_VEL
LIN {X 0,Y 151.036,Z 660.847,A -85,B 0,C 180,E1 -22560.772,E2 -22560.772} C_VEL
LIN {X 0,Y 146.743,Z 675.625,A -85,B 0,C 180,E1 -22562.587,E2 -22562.587} C_VEL
LIN {X 0,Y 140.968,Z 691.1,A -85,B 0,C 180,E1 -22565.257,E2 -22565.257} C_VEL
LIN {X 0,Y 134.859,Z 704.513,A -85,B 0,C 180,E1 -22568.465,E2 -22568.465} C_VEL
LIN {X 0,Y 128.291,Z 716.957,A -85,B 0,C 180,E1 -22572.534,E2 -22572.534} C_VEL
LIN {X 0,Y 121.953,Z 727.637,A -85,B 0,C 180,E1 -22577.337,E2 -22577.337} C_VEL
LIN {X 0,Y 115.623,Z 737.575,A -85,B 0,C 180,E1 -22583.54,E2 -22583.54} C_VEL
LIN {X 0,Y 110.526,Z 745.408,A -85,B 0,C 180,E1 -22590.513,E2 -22590.513} C_VEL
LIN {X 0,Y 106.76,Z 751.735,A -85,B 0,C 180,E1 -22598.612,E2 -22598.612} C_VEL
LIN {X 0,Y 104.797,Z 756.066,A -85,B 0,C 180,E1 -22607.197,E2 -22607.197} C_VEL
LIN {X 0,Y 104.379,Z 758.599,A -85,B 0,C 180,E1 -22615.779,E2 -22615.779} C_VEL
LIN {X 0,Y 105.213,Z 759.499,A -85,B 0,C 180,E1 -22624.227,E2 -22624.227} C_VEL
LIN {X 0,Y 107.995,Z 758.675,A -85,B 0,C 180,E1 -22633.236,E2 -22633.236} C_VEL
LIN {X 0,Y 112.72,Z 756.181,A -85,B 0,C 180,E1 -22641.304,E2 -22641.304} C_VEL
LIN {X 0,Y 119.467,Z 751.721,A -85,B 0,C 180,E1 -22648.74,E2 -22648.74} C_VEL
LIN {X 0,Y 127.342,Z 745.736,A -85,B 0,C 180,E1 -22654.911,E2 -22654.911} C_VEL
LIN {X 0,Y 136.408,Z 737.692,A -85,B 0,C 180,E1 -22660.293,E2 -22660.293} C_VEL
LIN {X 0,Y 145.802,Z 728.085,A -85,B 0,C 180,E1 -22664.687,E2 -22664.687} C_VEL
LIN {X 0,Y 154.519,Z 717.547,A -85,B 0,C 180,E1 -22668.048,E2 -22668.048} C_VEL
LIN {X 0,Y 163.036,Z 705.406,A -85,B 0,C 180,E1 -22670.855,E2 -22670.855} C_VEL
LIN {X 0,Y 170.624,Z 692.227,A -85,B 0,C 180,E1 -22673.055,E2 -22673.055} C_VEL
LIN {X 0,Y 177.363,Z 677.73,A -85,B 0,C 180,E1 -22674.824,E2 -22674.824} C_VEL
LIN {X 0,Y 182.738,Z 662.521,A -85,B 0,C 180,E1 -22676.157,E2 -22676.157} C_VEL
LIN {X 0,Y 186.878,Z 646.156,A -85,B 0,C 180,E1 -22677.154,E2 -22677.154} C_VEL
LIN {X 0,Y 189.47,Z 628.849,A -85,B 0,C 180,E1 -22677.813,E2 -22677.813} C_VEL
LIN {X 0,Y 200.876,Z 528.69,A -85,B 0,C 180,E1 -22680.516,E2 -22680.516} C_VEL
LIN {X 0,Y 202.968,Z 498.374,A -85,B 0,C 180,E1 -22683.105,E2 -22683.105} C_VEL
LIN {X 0,Y 203.464,Z 492.715,A -85,B 0,C 180,E1 -22683.662,E2 -22683.662} C_VEL
LIN {X 0,Y 212.252,Z 466.698,A -85,B 0,C 180,E1 -22686.626,E2 -22686.626} C_VEL
LIN {X 0,Y 212.753,Z 462.41,A -85,B 0,C 180,E1 -22689.74,E2 -22689.74} C_VEL
LIN {X 0,Y 213.323,Z 460.166,A -85,B 0,C 180,E1 -22692.45,E2 -22692.45} C_VEL
LIN {X 0,Y 213.55,Z 459.604,A -85,B 0,C 180,E1 -22693.719,E2 -22693.719} C_VEL
LIN {X 0,Y 206.277,Z 479.499,A -85,B 0,C 180,E1 -22694.773,E2 -22694.773} C_VEL
LIN {X 0,Y 200.62,Z 496.182,A -85,B 0,C 180,E1 -22695.754,E2 -22695.754} C_VEL
LIN {X 0,Y 196.225,Z 531.683,A -85,B 0,C 180,E1 -22696.899,E2 -22696.899} C_VEL
LIN {X 0,Y 192.277,Z 563.71,A -85,B 0,C 180,E1 -22697.966,E2 -22697.966} C_VEL
LIN {X 0,Y 191.222,Z 571.408,A -85,B 0,C 180,E1 -22697.93,E2 -22697.93} C_VEL
LIN {X 0,Y 188.028,Z 592.042,A -85,B 0,C 180,E1 -22696.695,E2 -22696.695} C_VEL
LIN {X 0,Y 187.137,Z 598.642,A -85,B 0,C 180,E1 -22696.697,E2 -22696.697} C_VEL
LIN {X 0,Y 181.549,Z 642.927,A -85,B 0,C 180,E1 -22698.579,E2 -22698.579} C_VEL
LIN {X 0,Y 178.106,Z 658.435,A -85,B 0,C 180,E1 -22699.49,E2 -22699.49} C_VEL
LIN {X 0,Y 173.62,Z 672.664,A -85,B 0,C 180,E1 -22700.605,E2 -22700.605} C_VEL
LIN {X 0,Y 167.783,Z 686.835,A -85,B 0,C 180,E1 -22702.091,E2 -22702.091} C_VEL
LIN {X 0,Y 160.423,Z 700.898,A -85,B 0,C 180,E1 -22704.077,E2 -22704.077} C_VEL
LIN {X 0,Y 151.679,Z 714.614,A -85,B 0,C 180,E1 -22706.732,E2 -22706.732} C_VEL
LIN {X 0,Y 142.874,Z 726.156,A -85,B 0,C 180,E1 -22709.809,E2 -22709.809} C_VEL
LIN {X 0,Y 132.777,Z 737.57,A -85,B 0,C 180,E1 -22714.081,E2 -22714.081} C_VEL
LIN {X 0,Y 123.517,Z 746.711,A -85,B 0,C 180,E1 -22719.012,E2 -22719.012} C_VEL
LIN {X 0,Y 114.193,Z 754.872,A -85,B 0,C 180,E1 -22725.544,E2 -22725.544} C_VEL
LIN {X 0,Y 106.548,Z 760.985,A -85,B 0,C 180,E1 -22733.096,E2 -22733.096} C_VEL
LIN {X 0,Y 100.347,Z 765.697,A -85,B 0,C 180,E1 -22742.727,E2 -22742.727} C_VEL
LIN {X 0,Y 97.203,Z 768.077,A -85,B 0,C 180,E1 -22752.033,E2 -22752.033} C_VEL
LIN {X 0,Y 96.247,Z 768.788,A -85,B 0,C 180,E1 -22761.644,E2 -22761.644} C_VEL
LIN {X 0,Y 96.485,Z 768.103,A -85,B 0,C 180,E1 -22769.413,E2 -22769.413} C_VEL
LIN {X 0,Y 96.408,Z 766.344,A -85,B 0,C 180,E1 -22776.557,E2 -22776.557} C_VEL
LIN {X 0,Y 97.352,Z 762.248,A -85,B 0,C 180,E1 -22786.106,E2 -22786.106} C_VEL
LIN {X 0,Y 98.808,Z 759.526,A -85,B 0,C 180,E1 -22791.06,E2 -22791.06} C_VEL
LIN {X 0,Y 106.5,Z 761.861,A -85,B 0,C 180,E1 -22806.268,E2 -22806.268} C_VEL
LIN {X 0,Y 120.177,Z 762.512,A -85,B 0,C 180,E1 -22818.274,E2 -22818.274} C_VEL
LIN {X 0,Y 106.854,Z 758.318,A -85,B 0,C 180,E1 -22829.651,E2 -22829.651} C_VEL
LIN {X 0,Y 99.417,Z 752.664,A -85,B 0,C 180,E1 -22842.441,E2 -22842.441} C_VEL
LIN {X 0,Y 96.969,Z 746.324,A -85,B 0,C 180,E1 -22854.084,E2 -22854.084} C_VEL
LIN {X 0,Y 96.615,Z 740.733,A -85,B 0,C 180,E1 -22862.375,E2 -22862.375} C_VEL
LIN {X 0,Y 97.166,Z 732.736,A -85,B 0,C 180,E1 -22871.879,E2 -22871.879} C_VEL
LIN {X 0,Y 99.565,Z 722.256,A -85,B 0,C 180,E1 -22881.814,E2 -22881.814} C_VEL
LIN {X 0,Y 103.846,Z 710.271,A -85,B 0,C 180,E1 -22890.686,E2 -22890.686} C_VEL
LIN {X 0,Y 110.06,Z 695.883,A -85,B 0,C 180,E1 -22898.82,E2 -22898.82} C_VEL
LIN {X 0,Y 118.936,Z 677.163,A -85,B 0,C 180,E1 -22906.829,E2 -22906.829} C_VEL
LIN {X 0,Y 120.78,Z 675.735,A -85,B 0,C 180,E1 -22908.166,E2 -22908.166} C_VEL
LIN {X 0,Y 124.934,Z 673.109,A -85,B 0,C 180,E1 -22910.204,E2 -22910.204} C_VEL
LIN {X 0,Y 130.437,Z 668.144,A -85,B 0,C 180,E1 -22912.146,E2 -22912.146} C_VEL
LIN {X 0,Y 137.482,Z 660.57,A -85,B 0,C 180,E1 -22914.187,E2 -22914.187} C_VEL
LIN {X 0,Y 142.414,Z 656.825,A -85,B 0,C 180,E1 -22915.943,E2 -22915.943} C_VEL
LIN {X 0,Y 148.096,Z 650.898,A -85,B 0,C 180,E1 -22917.539,E2 -22917.539} C_VEL
LIN {X 0,Y 144.107,Z 666.795,A -85,B 0,C 180,E1 -22919.103,E2 -22919.103} C_VEL
LIN {X 0,Y 139.079,Z 681.818,A -85,B 0,C 180,E1 -22921.201,E2 -22921.201} C_VEL
LIN {X 0,Y 132.823,Z 696.614,A -85,B 0,C 180,E1 -22924.107,E2 -22924.107} C_VEL
LIN {X 0,Y 126.221,Z 709.615,A -85,B 0,C 180,E1 -22927.647,E2 -22927.647} C_VEL
LIN {X 0,Y 118.94,Z 722.063,A -85,B 0,C 180,E1 -22932.379,E2 -22932.379} C_VEL
LIN {X 0,Y 112.445,Z 732.001,A -85,B 0,C 180,E1 -22937.672,E2 -22937.672} C_VEL
LIN {X 0,Y 106.079,Z 741.221,A -85,B 0,C 180,E1 -22944.586,E2 -22944.586} C_VEL
LIN {X 0,Y 101.226,Z 748.293,A -85,B 0,C 180,E1 -22952.258,E2 -22952.258} C_VEL
LIN {X 0,Y 97.873,Z 753.921,A -85,B 0,C 180,E1 -22961.256,E2 -22961.256} C_VEL
LIN {X 0,Y 96.521,Z 757.407,A -85,B 0,C 180,E1 -22969.982,E2 -22969.982} C_VEL
LIN {X 0,Y 96.537,Z 759.397,A -85,B 0,C 180,E1 -22979.122,E2 -22979.122} C_VEL
LIN {X 0,Y 98.131,Z 759.858,A -85,B 0,C 180,E1 -22988.419,E2 -22988.419} C_VEL
LIN {X 0,Y 101.812,Z 758.65,A -85,B 0,C 180,E1 -22997.428,E2 -22997.428} C_VEL
LIN {X 0,Y 108.18,Z 755.398,A -85,B 0,C 180,E1 -23006.318,E2 -23006.318} C_VEL
LIN {X 0,Y 116.08,Z 750.436,A -85,B 0,C 180,E1 -23013.599,E2 -23013.599} C_VEL
LIN {X 0,Y 125.614,Z 743.4,A -85,B 0,C 180,E1 -23019.91,E2 -23019.91} C_VEL
LIN {X 0,Y 134.821,Z 735.39,A -85,B 0,C 180,E1 -23024.581,E2 -23024.581} C_VEL
LIN {X 0,Y 144.8,Z 725.195,A -85,B 0,C 180,E1 -23028.648,E2 -23028.648} C_VEL
LIN {X 0,Y 153.602,Z 714.534,A -85,B 0,C 180,E1 -23031.63,E2 -23031.63} C_VEL
LIN {X 0,Y 162.092,Z 702.21,A -85,B 0,C 180,E1 -23034.121,E2 -23034.121} C_VEL
LIN {X 0,Y 169.85,Z 688.529,A -85,B 0,C 180,E1 -23036.129,E2 -23036.129} C_VEL
LIN {X 0,Y 176.597,Z 673.419,A -85,B 0,C 180,E1 -23037.727,E2 -23037.727} C_VEL
LIN {X 0,Y 181.755,Z 658.082,A -85,B 0,C 180,E1 -23038.888,E2 -23038.888} C_VEL
LIN {X 0,Y 185.599,Z 641.233,A -85,B 0,C 180,E1 -23039.751,E2 -23039.751} C_VEL
LIN {X 0,Y 189.124,Z 613.558,A -85,B 0,C 180,E1 -23040.571,E2 -23040.571} C_VEL
LIN {X 0,Y 198.993,Z 529.77,A -85,B 0,C 180,E1 -23042.735,E2 -23042.735} C_VEL
LIN {X 0,Y 201.501,Z 499.378,A -85,B 0,C 180,E1 -23045.355,E2 -23045.355} C_VEL
LIN {X 0,Y 202.492,Z 492.06,A -85,B 0,C 180,E1 -23046.093,E2 -23046.093} C_VEL
LIN {X 0,Y 209.424,Z 472.054,A -85,B 0,C 180,E1 -23048.372,E2 -23048.372} C_VEL
LIN {X 0,Y 210.157,Z 468.73,A -85,B 0,C 180,E1 -23051.248,E2 -23051.248} C_VEL
LIN {X 0,Y 210.313,Z 468.219,A -85,B 0,C 180,E1 -23052.012,E2 -23052.012} C_VEL
LIN {X 0,Y 200.315,Z 495.616,A -85,B 0,C 180,E1 -23053.395,E2 -23053.395} C_VEL
LIN {X 0,Y 197.502,Z 517.257,A -85,B 0,C 180,E1 -23054.154,E2 -23054.154} C_VEL
LIN {X 0,Y 188.057,Z 591.329,A -85,B 0,C 180,E1 -23056.458,E2 -23056.458} C_VEL
LIN {X 0,Y 187.137,Z 598.642,A -85,B 0,C 180,E1 -23056.697,E2 -23056.697} C_VEL
LIN {X 0,Y 186.104,Z 606.325,A -85,B 0,C 180,E1 -23056.694,E2 -23056.694} C_VEL
LIN {X 0,Y 183.049,Z 627.011,A -85,B 0,C 180,E1 -23055.602,E2 -23055.602} C_VEL
LIN {X 0,Y 182.139,Z 633.603,A -85,B 0,C 180,E1 -23055.605,E2 -23055.605} C_VEL
LIN {X 0,Y 179.13,Z 650.536,A -85,B 0,C 180,E1 -23056.405,E2 -23056.405} C_VEL
LIN {X 0,Y 174.484,Z 666.732,A -85,B 0,C 180,E1 -23057.44,E2 -23057.44} C_VEL
LIN {X 0,Y 168.449,Z 681.944,A -85,B 0,C 180,E1 -23058.798,E2 -23058.798} C_VEL
LIN {X 0,Y 160.342,Z 697.689,A -85,B 0,C 180,E1 -23060.726,E2 -23060.726} C_VEL
LIN {X 0,Y 151.57,Z 711.36,A -85,B 0,C 180,E1 -23063.052,E2 -23063.052} C_VEL
LIN {X 0,Y 141.459,Z 724.416,A -85,B 0,C 180,E1 -23066.159,E2 -23066.159} C_VEL
LIN {X 0,Y 131.424,Z 735.267,A -85,B 0,C 180,E1 -23069.865,E2 -23069.865} C_VEL
LIN {X 0,Y 121.323,Z 744.716,A -85,B 0,C 180,E1 -23074.51,E2 -23074.51} C_VEL
LIN {X 0,Y 111.521,Z 752.787,A -85,B 0,C 180,E1 -23080.361,E2 -23080.361} C_VEL
LIN {X 0,Y 102.063,Z 759.683,A -85,B 0,C 180,E1 -23088.237,E2 -23088.237} C_VEL
LIN {X 0,Y 95.159,Z 764.255,A -85,B 0,C 180,E1 -23096.89,E2 -23096.89} C_VEL
LIN {X 0,Y 90.167,Z 767.357,A -85,B 0,C 180,E1 -23107.858,E2 -23107.858} C_VEL
LIN {X 0,Y 88.358,Z 768.391,A -85,B 0,C 180,E1 -23118.255,E2 -23118.255} C_VEL
LIN {X 0,Y 88.417,Z 767.892,A -85,B 0,C 180,E1 -23127.414,E2 -23127.414} C_VEL
LIN {X 0,Y 88.438,Z 766.638,A -85,B 0,C 180,E1 -23133.897,E2 -23133.897} C_VEL
LIN {X 0,Y 88.885,Z 763.346,A -85,B 0,C 180,E1 -23143.671,E2 -23143.671} C_VEL
LIN {X 0,Y 91.828,Z 757.904,A -85,B 0,C 180,E1 -23154.106,E2 -23154.106} C_VEL
LIN {X 0,Y 101.042,Z 760.514,A -85,B 0,C 180,E1 -23170.039,E2 -23170.039} C_VEL
LIN {X 0,Y 110.236,Z 761.227,A -85,B 0,C 180,E1 -23178.258,E2 -23178.258} C_VEL
LIN {X 0,Y 97.038,Z 755.99,A -85,B 0,C 180,E1 -23191.155,E2 -23191.155} C_VEL
LIN {X 0,Y 90.694,Z 749.71,A -85,B 0,C 180,E1 -23204.66,E2 -23204.66} C_VEL
LIN {X 0,Y 88.962,Z 743.307,A -85,B 0,C 180,E1 -23216.136,E2 -23216.136} C_VEL
LIN {X 0,Y 88.758,Z 737.547,A -85,B 0,C 180,E1 -23224.525,E2 -23224.525} C_VEL
LIN {X 0,Y 89.716,Z 728.861,A -85,B 0,C 180,E1 -23234.855,E2 -23234.855} C_VEL
LIN {X 0,Y 92.715,Z 718.079,A -85,B 0,C 180,E1 -23245.044,E2 -23245.044} C_VEL
LIN {X 0,Y 97.747,Z 705.492,A -85,B 0,C 180,E1 -23254.238,E2 -23254.238} C_VEL
LIN {X 0,Y 103.832,Z 692.715,A -85,B 0,C 180,E1 -23261.643,E2 -23261.643} C_VEL
LIN {X 0,Y 105.291,Z 691.668,A -85,B 0,C 180,E1 -23263.138,E2 -23263.138} C_VEL
LIN {X 0,Y 109.019,Z 689.73,A -85,B 0,C 180,E1 -23265.676,E2 -23265.676} C_VEL
LIN {X 0,Y 115.039,Z 685.431,A -85,B 0,C 180,E1 -23268.374,E2 -23268.374} C_VEL
LIN {X 0,Y 118.258,Z 682.828,A -85,B 0,C 180,E1 -23269.55,E2 -23269.55} C_VEL
LIN {X 0,Y 122.432,Z 680.806,A -85,B 0,C 180,E1 -23271.631,E2 -23271.631} C_VEL
LIN {X 0,Y 128.761,Z 676.171,A -85,B 0,C 180,E1 -23273.864,E2 -23273.864} C_VEL
LIN {X 0,Y 138.249,Z 666.859,A -85,B 0,C 180,E1 -23276.278,E2 -23276.278} C_VEL
LIN {X 0,Y 139.018,Z 666.57,A -85,B 0,C 180,E1 -23276.598,E2 -23276.598} C_VEL
LIN {X 0,Y 133.704,Z 681.929,A -85,B 0,C 180,E1 -23278.711,E2 -23278.711} C_VEL
LIN {X 0,Y 127.234,Z 696.614,A -85,B 0,C 180,E1 -23281.582,E2 -23281.582} C_VEL
LIN {X 0,Y 120.594,Z 709.195,A -85,B 0,C 180,E1 -23284.98,E2 -23284.98} C_VEL
LIN {X 0,Y 112.859,Z 721.778,A -85,B 0,C 180,E1 -23289.781,E2 -23289.781} C_VEL
LIN {X 0,Y 105.907,Z 731.877,A -85,B 0,C 180,E1 -23295.226,E2 -23295.226} C_VEL
LIN {X 0,Y 99.024,Z 741.193,A -85,B 0,C 180,E1 -23302.451,E2 -23302.451} C_VEL
LIN {X 0,Y 93.722,Z 748.386,A -85,B 0,C 180,E1 -23310.605,E2 -23310.605} C_VEL
LIN {X 0,Y 90.043,Z 754.054,A -85,B 0,C 180,E1 -23320.227,E2 -23320.227} C_VEL
LIN {X 0,Y 88.531,Z 757.68,A -85,B 0,C 180,E1 -23329.797,E2 -23329.797} C_VEL
LIN {X 0,Y 88.573,Z 759.725,A -85,B 0,C 180,E1 -23339.627,E2 -23339.627} C_VEL
LIN {X 0,Y 90.6,Z 760.265,A -85,B 0,C 180,E1 -23350.402,E2 -23350.402} C_VEL
LIN {X 0,Y 94.993,Z 759,A -85,B 0,C 180,E1 -23360.197,E2 -23360.197} C_VEL
LIN {X 0,Y 102.174,Z 755.748,A -85,B 0,C 180,E1 -23369.433,E2 -23369.433} C_VEL
LIN {X 0,Y 110.419,Z 751.058,A -85,B 0,C 180,E1 -23376.518,E2 -23376.518} C_VEL
LIN {X 0,Y 120.399,Z 744.251,A -85,B 0,C 180,E1 -23382.731,E2 -23382.731} C_VEL
LIN {X 0,Y 130.125,Z 736.406,A -85,B 0,C 180,E1 -23387.357,E2 -23387.357} C_VEL
LIN {X 0,Y 140.571,Z 726.341,A -85,B 0,C 180,E1 -23391.338,E2 -23391.338} C_VEL
LIN {X 0,Y 150.194,Z 715.369,A -85,B 0,C 180,E1 -23394.356,E2 -23394.356} C_VEL
LIN {X 0,Y 159.215,Z 702.911,A -85,B 0,C 180,E1 -23396.786,E2 -23396.786} C_VEL
LIN {X 0,Y 167.011,Z 689.834,A -85,B 0,C 180,E1 -23398.634,E2 -23398.634} C_VEL
LIN {X 0,Y 173.615,Z 675.831,A -85,B 0,C 180,E1 -23400.077,E2 -23400.077} C_VEL
LIN {X 0,Y 179,Z 660.951,A -85,B 0,C 180,E1 -23401.193,E2 -23401.193} C_VEL
LIN {X 0,Y 183.01,Z 645.247,A -85,B 0,C 180,E1 -23402.014,E2 -23402.014} C_VEL
LIN {X 0,Y 185.876,Z 626.111,A -85,B 0,C 180,E1 -23402.634,E2 -23402.634} C_VEL
LIN {X 0,Y 197.404,Z 530.969,A -85,B 0,C 180,E1 -23404.984,E2 -23404.984} C_VEL
LIN {X 0,Y 200.381,Z 500.425,A -85,B 0,C 180,E1 -23407.633,E2 -23407.633} C_VEL
LIN {X 0,Y 201.509,Z 492.591,A -85,B 0,C 180,E1 -23408.416,E2 -23408.416} C_VEL
LIN {X 0,Y 206.852,Z 477.796,A -85,B 0,C 180,E1 -23410.02,E2 -23410.02} C_VEL
LIN {X 0,Y 206.855,Z 477.728,A -85,B 0,C 180,E1 -23410.204,E2 -23410.204} C_VEL
LIN {X 0,Y 200.331,Z 495.442,A -85,B 0,C 180,E1 -23411.054,E2 -23411.054} C_VEL
LIN {X 0,Y 198.215,Z 510.881,A -85,B 0,C 180,E1 -23411.654,E2 -23411.654} C_VEL
LIN {X 0,Y 189.294,Z 578.105,A -85,B 0,C 180,E1 -23413.673,E2 -23413.673} C_VEL
LIN {X 0,Y 185.604,Z 606.428,A -85,B 0,C 180,E1 -23414.553,E2 -23414.553} C_VEL
LIN {X 0,Y 182.139,Z 633.603,A -85,B 0,C 180,E1 -23415.605,E2 -23415.605} C_VEL
LIN {X 0,Y 180.92,Z 641.275,A -85,B 0,C 180,E1 -23415.54,E2 -23415.54} C_VEL
LIN {X 0,Y 176.871,Z 657.396,A -85,B 0,C 180,E1 -23414.739,E2 -23414.739} C_VEL
LIN {X 0,Y 174.09,Z 665.78,A -85,B 0,C 180,E1 -23414.747,E2 -23414.747} C_VEL
LIN {X 0,Y 173.374,Z 667.82,A -85,B 0,C 180,E1 -23414.855,E2 -23414.855} C_VEL
LIN {X 0,Y 166.583,Z 683.75,A -85,B 0,C 180,E1 -23416.205,E2 -23416.205} C_VEL
LIN {X 0,Y 158.64,Z 698.254,A -85,B 0,C 180,E1 -23417.895,E2 -23417.895} C_VEL
LIN {X 0,Y 149.523,Z 711.588,A -85,B 0,C 180,E1 -23420.043,E2 -23420.043} C_VEL
LIN {X 0,Y 138.97,Z 724.496,A -85,B 0,C 180,E1 -23422.951,E2 -23422.951} C_VEL
LIN {X 0,Y 128.415,Z 735.25,A -85,B 0,C 180,E1 -23426.452,E2 -23426.452} C_VEL
LIN {X 0,Y 117.666,Z 744.635,A -85,B 0,C 180,E1 -23430.892,E2 -23430.892} C_VEL
LIN {X 0,Y 107.08,Z 752.555,A -85,B 0,C 180,E1 -23436.591,E2 -23436.591} C_VEL
LIN {X 0,Y 96.662,Z 759.388,A -85,B 0,C 180,E1 -23444.471,E2 -23444.471} C_VEL
LIN {X 0,Y 88.83,Z 763.907,A -85,B 0,C 180,E1 -23453.385,E2 -23453.385} C_VEL
LIN {X 0,Y 82.896,Z 766.977,A -85,B 0,C 180,E1 -23465.038,E2 -23465.038} C_VEL
LIN {X 0,Y 80.502,Z 767.97,A -85,B 0,C 180,E1 -23476.358,E2 -23476.358} C_VEL
LIN {X 0,Y 80.39,Z 767.466,A -85,B 0,C 180,E1 -23486.442,E2 -23486.442} C_VEL
LIN {X 0,Y 80.473,Z 766.373,A -85,B 0,C 180,E1 -23492.856,E2 -23492.856} C_VEL
LIN {X 0,Y 80.766,Z 763.426,A -85,B 0,C 180,E1 -23502.883,E2 -23502.883} C_VEL
LIN {X 0,Y 83.246,Z 758.568,A -85,B 0,C 180,E1 -23513.358,E2 -23513.358} C_VEL
LIN {X 0,Y 85.166,Z 756.173,A -85,B 0,C 180,E1 -23517.636,E2 -23517.636} C_VEL
LIN {X 0,Y 96.108,Z 758.934,A -85,B 0,C 180,E1 -23534.198,E2 -23534.198} C_VEL
LIN {X 0,Y 100.46,Z 759.439,A -85,B 0,C 180,E1 -23538.179,E2 -23538.179} C_VEL
LIN {X 0,Y 87.854,Z 753.433,A -85,B 0,C 180,E1 -23552.187,E2 -23552.187} C_VEL
LIN {X 0,Y 82.289,Z 746.59,A -85,B 0,C 180,E1 -23566.655,E2 -23566.655} C_VEL
LIN {X 0,Y 81.03,Z 740.337,A -85,B 0,C 180,E1 -23577.881,E2 -23577.881} C_VEL
LIN {X 0,Y 81.014,Z 733.468,A -85,B 0,C 180,E1 -23587.805,E2 -23587.805} C_VEL
LIN {X 0,Y 82.679,Z 723.905,A -85,B 0,C 180,E1 -23599.06,E2 -23599.06} C_VEL
LIN {X 0,Y 86.675,Z 712.325,A -85,B 0,C 180,E1 -23609.741,E2 -23609.741} C_VEL
LIN {X 0,Y 89.909,Z 705.194,A -85,B 0,C 180,E1 -23615.333,E2 -23615.333} C_VEL
LIN {X 0,Y 93.73,Z 703.212,A -85,B 0,C 180,E1 -23619.798,E2 -23619.798} C_VEL
LIN {X 0,Y 99.145,Z 700.001,A -85,B 0,C 180,E1 -23623.299,E2 -23623.299} C_VEL
LIN {X 0,Y 101.986,Z 698.217,A -85,B 0,C 180,E1 -23624.903,E2 -23624.903} C_VEL
LIN {X 0,Y 106.526,Z 696.253,A -85,B 0,C 180,E1 -23627.863,E2 -23627.863} C_VEL
LIN {X 0,Y 112.676,Z 692.477,A -85,B 0,C 180,E1 -23630.539,E2 -23630.539} C_VEL
LIN {X 0,Y 117.65,Z 688.952,A -85,B 0,C 180,E1 -23632.223,E2 -23632.223} C_VEL
LIN {X 0,Y 122.934,Z 686.293,A -85,B 0,C 180,E1 -23634.426,E2 -23634.426} C_VEL
LIN {X 0,Y 128.274,Z 682.808,A -85,B 0,C 180,E1 -23636.147,E2 -23636.147} C_VEL
LIN {X 0,Y 121.466,Z 697.509,A -85,B 0,C 180,E1 -23639.032,E2 -23639.032} C_VEL
LIN {X 0,Y 114.185,Z 710.484,A -85,B 0,C 180,E1 -23642.626,E2 -23642.626} C_VEL
LIN {X 0,Y 106.384,Z 722.448,A -85,B 0,C 180,E1 -23647.329,E2 -23647.329} C_VEL
LIN {X 0,Y 99.006,Z 732.483,A -85,B 0,C 180,E1 -23652.964,E2 -23652.964} C_VEL
LIN {X 0,Y 91.654,Z 741.765,A -85,B 0,C 180,E1 -23660.575,E2 -23660.575} C_VEL
LIN {X 0,Y 85.964,Z 748.909,A -85,B 0,C 180,E1 -23669.326,E2 -23669.326} C_VEL
LIN {X 0,Y 82.037,Z 754.55,A -85,B 0,C 180,E1 -23679.817,E2 -23679.817} C_VEL
LIN {X 0,Y 80.493,Z 758.137,A -85,B 0,C 180,E1 -23690.345,E2 -23690.345} C_VEL
LIN {X 0,Y 80.643,Z 760.087,A -85,B 0,C 180,E1 -23700.544,E2 -23700.544} C_VEL
LIN {X 0,Y 83.067,Z 760.678,A -85,B 0,C 180,E1 -23712.37,E2 -23712.37} C_VEL
LIN {X 0,Y 88.241,Z 759.445,A -85,B 0,C 180,E1 -23723.088,E2 -23723.088} C_VEL
LIN {X 0,Y 96.441,Z 756.144,A -85,B 0,C 180,E1 -23732.857,E2 -23732.857} C_VEL
LIN {X 0,Y 105.534,Z 751.404,A -85,B 0,C 180,E1 -23740.056,E2 -23740.056} C_VEL
LIN {X 0,Y 116.327,Z 744.542,A -85,B 0,C 180,E1 -23746.205,E2 -23746.205} C_VEL
LIN {X 0,Y 126.642,Z 736.699,A -85,B 0,C 180,E1 -23750.679,E2 -23750.679} C_VEL
LIN {X 0,Y 137.608,Z 726.695,A -85,B 0,C 180,E1 -23754.47,E2 -23754.47} C_VEL
LIN {X 0,Y 147.467,Z 715.938,A -85,B 0,C 180,E1 -23757.278,E2 -23757.278} C_VEL
LIN {X 0,Y 157.117,Z 703.061,A -85,B 0,C 180,E1 -23759.634,E2 -23759.634} C_VEL
LIN {X 0,Y 165.295,Z 689.668,A -85,B 0,C 180,E1 -23761.385,E2 -23761.385} C_VEL
LIN {X 0,Y 172.16,Z 675.328,A -85,B 0,C 180,E1 -23762.742,E2 -23762.742} C_VEL
LIN {X 0,Y 177.62,Z 660.411,A -85,B 0,C 180,E1 -23763.766,E2 -23763.766} C_VEL
LIN {X 0,Y 181.652,Z 644.499,A -85,B 0,C 180,E1 -23764.523,E2 -23764.523} C_VEL
LIN {X 0,Y 184.606,Z 624.815,A -85,B 0,C 180,E1 -23765.106,E2 -23765.106} C_VEL
LIN {X 0,Y 196.284,Z 532.135,A -85,B 0,C 180,E1 -23767.275,E2 -23767.275} C_VEL
LIN {X 0,Y 198.811,Z 508.879,A -85,B 0,C 180,E1 -23769.274,E2 -23769.274} C_VEL
LIN {X 0,Y 188.972,Z 579.992,A -85,B 0,C 180,E1 -23771.299,E2 -23771.299} C_VEL
LIN {X 0,Y 185.287,Z 607.063,A -85,B 0,C 180,E1 -23772.086,E2 -23772.086} C_VEL
LIN {X 0,Y 180.198,Z 643.184,A -85,B 0,C 180,E1 -23773.475,E2 -23773.475} C_VEL
LIN {X 0,Y 176.075,Z 659.703,A -85,B 0,C 180,E1 -23774.342,E2 -23774.342} C_VEL
LIN {X 0,Y 173.374,Z 667.82,A -85,B 0,C 180,E1 -23774.855,E2 -23774.855} C_VEL
LIN {X 0,Y 170.527,Z 675.034,A -85,B 0,C 180,E1 -23775.052,E2 -23775.052} C_VEL
LIN {X 0,Y 162.893,Z 689.903,A -85,B 0,C 180,E1 -23774.674,E2 -23774.674} C_VEL
LIN {X 0,Y 158.251,Z 697.43,A -85,B 0,C 180,E1 -23774.878,E2 -23774.878} C_VEL
LIN {X 0,Y 157.068,Z 699.223,A -85,B 0,C 180,E1 -23775.061,E2 -23775.061} C_VEL
LIN {X 0,Y 147.018,Z 713.143,A -85,B 0,C 180,E1 -23777.168,E2 -23777.168} C_VEL
LIN {X 0,Y 136.938,Z 724.638,A -85,B 0,C 180,E1 -23779.643,E2 -23779.643} C_VEL
LIN {X 0,Y 125.676,Z 735.412,A -85,B 0,C 180,E1 -23782.943,E2 -23782.943} C_VEL
LIN {X 0,Y 114.499,Z 744.553,A -85,B 0,C 180,E1 -23787.05,E2 -23787.05} C_VEL
LIN {X 0,Y 103.147,Z 752.381,A -85,B 0,C 180,E1 -23792.518,E2 -23792.518} C_VEL
LIN {X 0,Y 91.726,Z 759.126,A -85,B 0,C 180,E1 -23800.279,E2 -23800.279} C_VEL
LIN {X 0,Y 82.399,Z 763.775,A -85,B 0,C 180,E1 -23809.986,E2 -23809.986} C_VEL
LIN {X 0,Y 75.86,Z 766.598,A -85,B 0,C 180,E1 -23821.683,E2 -23821.683} C_VEL
LIN {X 0,Y 72.641,Z 767.542,A -85,B 0,C 180,E1 -23834.849,E2 -23834.849} C_VEL
LIN {X 0,Y 72.425,Z 766.832,A -85,B 0,C 180,E1 -23846.843,E2 -23846.843} C_VEL
LIN {X 0,Y 72.478,Z 765.784,A -85,B 0,C 180,E1 -23853.172,E2 -23853.172} C_VEL
LIN {X 0,Y 72.915,Z 762.719,A -85,B 0,C 180,E1 -23864.298,E2 -23864.298} C_VEL
LIN {X 0,Y 75.889,Z 757.673,A -85,B 0,C 180,E1 -23875.78,E2 -23875.78} C_VEL
LIN {X 0,Y 78.9,Z 754.318,A -85,B 0,C 180,E1 -23881.738,E2 -23881.738} C_VEL
LIN {X 0,Y 90.825,Z 757.158,A -85,B 0,C 180,E1 -23898.052,E2 -23898.052} C_VEL
LIN {X 0,Y 78.705,Z 750.338,A -85,B 0,C 180,E1 -23913.603,E2 -23913.603} C_VEL
LIN {X 0,Y 74.013,Z 743.023,A -85,B 0,C 180,E1 -23929.101,E2 -23929.101} C_VEL
LIN {X 0,Y 73.132,Z 736.982,A -85,B 0,C 180,E1 -23940.003,E2 -23940.003} C_VEL
LIN {X 0,Y 73.439,Z 729.182,A -85,B 0,C 180,E1 -23951.361,E2 -23951.361} C_VEL
LIN {X 0,Y 75.876,Z 719.073,A -85,B 0,C 180,E1 -23963.289,E2 -23963.289} C_VEL
LIN {X 0,Y 77.262,Z 715.627,A -85,B 0,C 180,E1 -23967.352,E2 -23967.352} C_VEL
LIN {X 0,Y 80.016,Z 714.206,A -85,B 0,C 180,E1 -23972.504,E2 -23972.504} C_VEL
LIN {X 0,Y 85.277,Z 711.198,A -85,B 0,C 180,E1 -23977.57,E2 -23977.57} C_VEL
LIN {X 0,Y 87.014,Z 710.408,A -85,B 0,C 180,E1 -23979.2,E2 -23979.2} C_VEL
LIN {X 0,Y 91.723,Z 708.571,A -85,B 0,C 180,E1 -23983.377,E2 -23983.377} C_VEL
LIN {X 0,Y 99.196,Z 704.36,A -85,B 0,C 180,E1 -23987.379,E2 -23987.379} C_VEL
LIN {X 0,Y 104.742,Z 702.123,A -85,B 0,C 180,E1 -23990.647,E2 -23990.647} C_VEL
LIN {X 0,Y 112.023,Z 698.059,A -85,B 0,C 180,E1 -23993.449,E2 -23993.449} C_VEL
LIN {X 0,Y 117.176,Z 694.798,A -85,B 0,C 180,E1 -23995.004,E2 -23995.004} C_VEL
LIN {X 0,Y 117.963,Z 694.596,A -85,B 0,C 180,E1 -23995.391,E2 -23995.391} C_VEL
LIN {X 0,Y 109.975,Z 708.678,A -85,B 0,C 180,E1 -23998.992,E2 -23998.992} C_VEL
LIN {X 0,Y 102.217,Z 720.24,A -85,B 0,C 180,E1 -24003.252,E2 -24003.252} C_VEL
LIN {X 0,Y 93.527,Z 731.572,A -85,B 0,C 180,E1 -24009.335,E2 -24009.335} C_VEL
LIN {X 0,Y 85.954,Z 740.513,A -85,B 0,C 180,E1 -24016.54,E2 -24016.54} C_VEL
LIN {X 0,Y 79.179,Z 748.334,A -85,B 0,C 180,E1 -24026.065,E2 -24026.065} C_VEL
LIN {X 0,Y 74.669,Z 754.044,A -85,B 0,C 180,E1 -24036.913,E2 -24036.913} C_VEL
LIN {X 0,Y 72.552,Z 758.154,A -85,B 0,C 180,E1 -24049.305,E2 -24049.305} C_VEL
LIN {X 0,Y 72.636,Z 760.318,A -85,B 0,C 180,E1 -24060.608,E2 -24060.608} C_VEL
LIN {X 0,Y 75.016,Z 761.116,A -85,B 0,C 180,E1 -24072.851,E2 -24072.851} C_VEL
LIN {X 0,Y 80.68,Z 760.183,A -85,B 0,C 180,E1 -24084.863,E2 -24084.863} C_VEL
LIN {X 0,Y 88.875,Z 757.43,A -85,B 0,C 180,E1 -24094.688,E2 -24094.688} C_VEL
LIN {X 0,Y 99.392,Z 752.664,A -85,B 0,C 180,E1 -24102.854,E2 -24102.854} C_VEL
LIN {X 0,Y 110.101,Z 746.582,A -85,B 0,C 180,E1 -24108.716,E2 -24108.716} C_VEL
LIN {X 0,Y 121.751,Z 738.511,A -85,B 0,C 180,E1 -24113.508,E2 -24113.508} C_VEL
LIN {X 0,Y 132.424,Z 729.588,A -85,B 0,C 180,E1 -24116.969,E2 -24116.969} C_VEL
LIN {X 0,Y 143.517,Z 718.31,A -85,B 0,C 180,E1 -24119.916,E2 -24119.916} C_VEL
LIN {X 0,Y 153.065,Z 706.554,A -85,B 0,C 180,E1 -24122.063,E2 -24122.063} C_VEL
LIN {X 0,Y 162.337,Z 692.374,A -85,B 0,C 180,E1 -24123.887,E2 -24123.887} C_VEL
LIN {X 0,Y 169.658,Z 678.327,A -85,B 0,C 180,E1 -24125.188,E2 -24125.188} C_VEL
LIN {X 0,Y 175.677,Z 663.027,A -85,B 0,C 180,E1 -24126.207,E2 -24126.207} C_VEL
LIN {X 0,Y 180.127,Z 647.184,A -85,B 0,C 180,E1 -24126.946,E2 -24126.946} C_VEL
LIN {X 0,Y 183.131,Z 629.093,A -85,B 0,C 180,E1 -24127.485,E2 -24127.485} C_VEL
LIN {X 0,Y 190.142,Z 574.635,A -85,B 0,C 180,E1 -24128.688,E2 -24128.688} C_VEL
LIN {X 0,Y 185.241,Z 609.39,A -85,B 0,C 180,E1 -24129.689,E2 -24129.689} C_VEL
LIN {X 0,Y 180.208,Z 642.95,A -85,B 0,C 180,E1 -24130.891,E2 -24130.891} C_VEL
LIN {X 0,Y 175.745,Z 659.909,A -85,B 0,C 180,E1 -24131.709,E2 -24131.709} C_VEL
LIN {X 0,Y 170.109,Z 674.932,A -85,B 0,C 180,E1 -24132.676,E2 -24132.676} C_VEL
LIN {X 0,Y 162.33,Z 690.556,A -85,B 0,C 180,E1 -24134.063,E2 -24134.063} C_VEL
LIN {X 0,Y 157.068,Z 699.223,A -85,B 0,C 180,E1 -24135.061,E2 -24135.061} C_VEL
LIN {X 0,Y 152.613,Z 705.586,A -85,B 0,C 180,E1 -24135.527,E2 -24135.527} C_VEL
LIN {X 0,Y 141.802,Z 718.379,A -85,B 0,C 180,E1 -24135.657,E2 -24135.657} C_VEL
LIN {X 0,Y 135.709,Z 724.556,A -85,B 0,C 180,E1 -24136.219,E2 -24136.219} C_VEL
LIN {X 0,Y 134.224,Z 725.992,A -85,B 0,C 180,E1 -24136.513,E2 -24136.513} C_VEL
LIN {X 0,Y 122.691,Z 736.321,A -85,B 0,C 180,E1 -24139.518,E2 -24139.518} C_VEL
LIN {X 0,Y 110.223,Z 745.581,A -85,B 0,C 180,E1 -24143.64,E2 -24143.64} C_VEL
LIN {X 0,Y 97.48,Z 753.566,A -85,B 0,C 180,E1 -24149.34,E2 -24149.34} C_VEL
LIN {X 0,Y 85.991,Z 759.5,A -85,B 0,C 180,E1 -24156.663,E2 -24156.663} C_VEL
LIN {X 0,Y 75.778,Z 763.884,A -85,B 0,C 180,E1 -24166.688,E2 -24166.688} C_VEL
LIN {X 0,Y 68.438,Z 766.402,A -85,B 0,C 180,E1 -24179.258,E2 -24179.258} C_VEL
LIN {X 0,Y 64.726,Z 767.11,A -85,B 0,C 180,E1 -24193.866,E2 -24193.866} C_VEL
LIN {X 0,Y 64.428,Z 766.293,A -85,B 0,C 180,E1 -24206.451,E2 -24206.451} C_VEL
LIN {X 0,Y 64.482,Z 765.187,A -85,B 0,C 180,E1 -24213.566,E2 -24213.566} C_VEL
LIN {X 0,Y 65.116,Z 761.97,A -85,B 0,C 180,E1 -24226.055,E2 -24226.055} C_VEL
LIN {X 0,Y 69.056,Z 756.343,A -85,B 0,C 180,E1 -24239.501,E2 -24239.501} C_VEL
LIN {X 0,Y 73.135,Z 752.298,A -85,B 0,C 180,E1 -24246.502,E2 -24246.502} C_VEL
LIN {X 0,Y 81.293,Z 754.38,A -85,B 0,C 180,E1 -24257.911,E2 -24257.911} C_VEL
LIN {X 0,Y 69.996,Z 747.071,A -85,B 0,C 180,E1 -24274.629,E2 -24274.629} C_VEL
LIN {X 0,Y 66.064,Z 739.825,A -85,B 0,C 180,E1 -24290.42,E2 -24290.42} C_VEL
LIN {X 0,Y 65.329,Z 734.226,A -85,B 0,C 180,E1 -24300.88,E2 -24300.88} C_VEL
LIN {X 0,Y 65.969,Z 725.345,A -85,B 0,C 180,E1 -24314.935,E2 -24314.935} C_VEL
LIN {X 0,Y 68.122,Z 723.565,A -85,B 0,C 180,E1 -24323.35,E2 -24323.35} C_VEL
LIN {X 0,Y 72.331,Z 721.023,A -85,B 0,C 180,E1 -24329.848,E2 -24329.848} C_VEL
LIN {X 0,Y 75.822,Z 719.697,A -85,B 0,C 180,E1 -24335.47,E2 -24335.47} C_VEL
LIN {X 0,Y 82.187,Z 716.544,A -85,B 0,C 180,E1 -24341.071,E2 -24341.071} C_VEL
LIN {X 0,Y 89.21,Z 713.971,A -85,B 0,C 180,E1 -24346.766,E2 -24346.766} C_VEL
LIN {X 0,Y 97.089,Z 710.026,A -85,B 0,C 180,E1 -24350.572,E2 -24350.572} C_VEL
LIN {X 0,Y 103.855,Z 707.383,A -85,B 0,C 180,E1 -24353.973,E2 -24353.973} C_VEL
LIN {X 0,Y 106.393,Z 706.31,A -85,B 0,C 180,E1 -24355.015,E2 -24355.015} C_VEL
LIN {X 0,Y 97.549,Z 719.192,A -85,B 0,C 180,E1 -24359.432,E2 -24359.432} C_VEL
LIN {X 0,Y 89.15,Z 729.674,A -85,B 0,C 180,E1 -24364.767,E2 -24364.767} C_VEL
LIN {X 0,Y 80.731,Z 739.119,A -85,B 0,C 180,E1 -24371.955,E2 -24371.955} C_VEL
LIN {X 0,Y 73.695,Z 746.58,A -85,B 0,C 180,E1 -24380.621,E2 -24380.621} C_VEL
LIN {X 0,Y 67.814,Z 753.089,A -85,B 0,C 180,E1 -24392.526,E2 -24392.526} C_VEL
LIN {X 0,Y 64.921,Z 757.44,A -85,B 0,C 180,E1 -24405.168,E2 -24405.168} C_VEL
LIN {X 0,Y 64.45,Z 760.077,A -85,B 0,C 180,E1 -24417.829,E2 -24417.829} C_VEL
LIN {X 0,Y 66.412,Z 761.418,A -85,B 0,C 180,E1 -24431.472,E2 -24431.472} C_VEL
LIN {X 0,Y 71.987,Z 761.119,A -85,B 0,C 180,E1 -24445.016,E2 -24445.016} C_VEL
LIN {X 0,Y 80.809,Z 758.834,A -85,B 0,C 180,E1 -24456.272,E2 -24456.272} C_VEL
LIN {X 0,Y 91.592,Z 754.786,A -85,B 0,C 180,E1 -24464.809,E2 -24464.809} C_VEL
LIN {X 0,Y 103.211,Z 749.027,A -85,B 0,C 180,E1 -24471.119,E2 -24471.119} C_VEL
LIN {X 0,Y 115.589,Z 741.414,A -85,B 0,C 180,E1 -24476.03,E2 -24476.03} C_VEL
LIN {X 0,Y 127.033,Z 732.691,A -85,B 0,C 180,E1 -24479.547,E2 -24479.547} C_VEL
LIN {X 0,Y 139.102,Z 721.545,A -85,B 0,C 180,E1 -24482.519,E2 -24482.519} C_VEL
LIN {X 0,Y 149.898,Z 709.196,A -85,B 0,C 180,E1 -24484.733,E2 -24484.733} C_VEL
LIN {X 0,Y 158.934,Z 696.533,A -85,B 0,C 180,E1 -24486.332,E2 -24486.332} C_VEL
LIN {X 0,Y 167.103,Z 682.021,A -85,B 0,C 180,E1 -24487.645,E2 -24487.645} C_VEL
LIN {X 0,Y 173.545,Z 667.21,A -85,B 0,C 180,E1 -24488.614,E2 -24488.614} C_VEL
LIN {X 0,Y 176.21,Z 659.357,A -85,B 0,C 180,E1 -24489.034,E2 -24489.034} C_VEL
LIN {X 0,Y 170.487,Z 674.177,A -85,B 0,C 180,E1 -24489.872,E2 -24489.872} C_VEL
LIN {X 0,Y 162.496,Z 689.733,A -85,B 0,C 180,E1 -24491.085,E2 -24491.085} C_VEL
LIN {X 0,Y 153.174,Z 704.064,A -85,B 0,C 180,E1 -24492.633,E2 -24492.633} C_VEL
LIN {X 0,Y 142.145,Z 717.745,A -85,B 0,C 180,E1 -24494.739,E2 -24494.739} C_VEL
LIN {X 0,Y 134.224,Z 725.992,A -85,B 0,C 180,E1 -24496.513,E2 -24496.513} C_VEL
LIN {X 0,Y 128.623,Z 731.089,A -85,B 0,C 180,E1 -24497.367,E2 -24497.367} C_VEL
LIN {X 0,Y 116.138,Z 740.451,A -85,B 0,C 180,E1 -24498.18,E2 -24498.18} C_VEL
LIN {X 0,Y 108.922,Z 745.09,A -85,B 0,C 180,E1 -24499.24,E2 -24499.24} C_VEL
LIN {X 0,Y 106.387,Z 746.675,A -85,B 0,C 180,E1 -24499.969,E2 -24499.969} C_VEL
LIN {X 0,Y 93.756,Z 753.811,A -85,B 0,C 180,E1 -24504.994,E2 -24504.994} C_VEL
LIN {X 0,Y 80.647,Z 759.857,A -85,B 0,C 180,E1 -24512.55,E2 -24512.55} C_VEL
LIN {X 0,Y 69.454,Z 763.951,A -85,B 0,C 180,E1 -24522.775,E2 -24522.775} C_VEL
LIN {X 0,Y 60.793,Z 766.268,A -85,B 0,C 180,E1 -24537.142,E2 -24537.142} C_VEL
LIN {X 0,Y 56.725,Z 766.625,A -85,B 0,C 180,E1 -24553.631,E2 -24553.631} C_VEL
LIN {X 0,Y 56.508,Z 765.497,A -85,B 0,C 180,E1 -24567.983,E2 -24567.983} C_VEL
LIN {X 0,Y 56.474,Z 763.867,A -85,B 0,C 180,E1 -24577.515,E2 -24577.515} C_VEL
LIN {X 0,Y 58.195,Z 759.958,A -85,B 0,C 180,E1 -24592.22,E2 -24592.22} C_VEL
LIN {X 0,Y 63.488,Z 754.1,A -85,B 0,C 180,E1 -24605.653,E2 -24605.653} C_VEL
LIN {X 0,Y 68.116,Z 750.143,A -85,B 0,C 180,E1 -24612.199,E2 -24612.199} C_VEL
LIN {X 0,Y 71.993,Z 751.186,A -85,B 0,C 180,E1 -24617.606,E2 -24617.606} C_VEL
LIN {X 0,Y 61.378,Z 743.366,A -85,B 0,C 180,E1 -24635.971,E2 -24635.971} C_VEL
LIN {X 0,Y 58.154,Z 736.312,A -85,B 0,C 180,E1 -24652.098,E2 -24652.098} C_VEL
LIN {X 0,Y 57.519,Z 734.41,A -85,B 0,C 180,E1 -24658.011,E2 -24658.011} C_VEL
LIN {X 0,Y 58.411,Z 731.695,A -85,B 0,C 180,E1 -24671.857,E2 -24671.857} C_VEL
LIN {X 0,Y 60.125,Z 730.132,A -85,B 0,C 180,E1 -24677.421,E2 -24677.421} C_VEL
LIN {X 0,Y 62.947,Z 728.562,A -85,B 0,C 180,E1 -24686.412,E2 -24686.412} C_VEL
LIN {X 0,Y 67.604,Z 726.252,A -85,B 0,C 180,E1 -24693.181,E2 -24693.181} C_VEL
LIN {X 0,Y 72.235,Z 724.628,A -85,B 0,C 180,E1 -24699.552,E2 -24699.552} C_VEL
LIN {X 0,Y 79.823,Z 721.449,A -85,B 0,C 180,E1 -24705.564,E2 -24705.564} C_VEL
LIN {X 0,Y 86.103,Z 719.412,A -85,B 0,C 180,E1 -24710.037,E2 -24710.037} C_VEL
LIN {X 0,Y 95.461,Z 715.31,A -85,B 0,C 180,E1 -24714.205,E2 -24714.205} C_VEL
LIN {X 0,Y 85.963,Z 727.021,A -85,B 0,C 180,E1 -24719.402,E2 -24719.402} C_VEL
LIN {X 0,Y 76.762,Z 736.948,A -85,B 0,C 180,E1 -24726.176,E2 -24726.176} C_VEL
LIN {X 0,Y 68.066,Z 745.467,A -85,B 0,C 180,E1 -24735.53,E2 -24735.53} C_VEL
LIN {X 0,Y 61.42,Z 752.029,A -85,B 0,C 180,E1 -24747.191,E2 -24747.191} C_VEL
LIN {X 0,Y 57.272,Z 757.066,A -85,B 0,C 180,E1 -24762.119,E2 -24762.119} C_VEL
LIN {X 0,Y 56.402,Z 759.99,A -85,B 0,C 180,E1 -24776.295,E2 -24776.295} C_VEL
LIN {X 0,Y 58.328,Z 761.709,A -85,B 0,C 180,E1 -24791.939,E2 -24791.939} C_VEL
LIN {X 0,Y 64.301,Z 761.713,A -85,B 0,C 180,E1 -24807.087,E2 -24807.087} C_VEL
LIN {X 0,Y 73.795,Z 759.875,A -85,B 0,C 180,E1 -24819.184,E2 -24819.184} C_VEL
LIN {X 0,Y 85.758,Z 755.977,A -85,B 0,C 180,E1 -24828.299,E2 -24828.299} C_VEL
LIN {X 0,Y 97.46,Z 750.884,A -85,B 0,C 180,E1 -24834.277,E2 -24834.277} C_VEL
LIN {X 0,Y 110.023,Z 743.873,A -85,B 0,C 180,E1 -24838.957,E2 -24838.957} C_VEL
LIN {X 0,Y 122.076,Z 735.631,A -85,B 0,C 180,E1 -24842.386,E2 -24842.386} C_VEL
LIN {X 0,Y 133.472,Z 726.12,A -85,B 0,C 180,E1 -24844.978,E2 -24844.978} C_VEL
LIN {X 0,Y 145.103,Z 714.153,A -85,B 0,C 180,E1 -24847.175,E2 -24847.175} C_VEL
LIN {X 0,Y 154.758,Z 701.944,A -85,B 0,C 180,E1 -24848.729,E2 -24848.729} C_VEL
LIN {X 0,Y 156.744,Z 699.029,A -85,B 0,C 180,E1 -24849.054,E2 -24849.054} C_VEL
LIN {X 0,Y 146.94,Z 711.745,A -85,B 0,C 180,E1 -24850.526,E2 -24850.526} C_VEL
LIN {X 0,Y 136.148,Z 723.337,A -85,B 0,C 180,E1 -24852.406,E2 -24852.406} C_VEL
LIN {X 0,Y 123.255,Z 734.735,A -85,B 0,C 180,E1 -24855.151,E2 -24855.151} C_VEL
LIN {X 0,Y 110.726,Z 743.904,A -85,B 0,C 180,E1 -24858.551,E2 -24858.551} C_VEL
LIN {X 0,Y 106.387,Z 746.675,A -85,B 0,C 180,E1 -24859.969,E2 -24859.969} C_VEL
LIN {X 0,Y 100.144,Z 750.256,A -85,B 0,C 180,E1 -24861.597,E2 -24861.597} C_VEL
LIN {X 0,Y 86.261,Z 756.396,A -85,B 0,C 180,E1 -24864.004,E2 -24864.004} C_VEL
LIN {X 0,Y 78.541,Z 759.227,A -85,B 0,C 180,E1 -24866.378,E2 -24866.378} C_VEL
LIN {X 0,Y 75.947,Z 760.138,A -85,B 0,C 180,E1 -24867.77,E2 -24867.77} C_VEL
LIN {X 0,Y 62.872,Z 764.131,A -85,B 0,C 180,E1 -24878.825,E2 -24878.825} C_VEL
LIN {X 0,Y 53.676,Z 766.019,A -85,B 0,C 180,E1 -24893.425,E2 -24893.425} C_VEL
LIN {X 0,Y 48.85,Z 766.079,A -85,B 0,C 180,E1 -24912.134,E2 -24912.134} C_VEL
LIN {X 0,Y 48.562,Z 764.748,A -85,B 0,C 180,E1 -24928.833,E2 -24928.833} C_VEL
LIN {X 0,Y 48.632,Z 762.584,A -85,B 0,C 180,E1 -24941.877,E2 -24941.877} C_VEL
LIN {X 0,Y 52.117,Z 757.693,A -85,B 0,C 180,E1 -24959.935,E2 -24959.935} C_VEL
LIN {X 0,Y 58.828,Z 751.676,A -85,B 0,C 180,E1 -24972.846,E2 -24972.846} C_VEL
LIN {X 0,Y 62.413,Z 748.566,A -85,B 0,C 180,E1 -24977.406,E2 -24977.406} C_VEL
LIN {X 0,Y 51.174,Z 741.184,A -85,B 0,C 180,E1 -25007.722,E2 -25007.722} C_VEL
LIN {X 0,Y 51.024,Z 739.137,A -85,B 0,C 180,E1 -25016.634,E2 -25016.634} C_VEL
LIN {X 0,Y 52.296,Z 736.24,A -85,B 0,C 180,E1 -25034.396,E2 -25034.396} C_VEL
LIN {X 0,Y 54.257,Z 734.849,A -85,B 0,C 180,E1 -25040.5,E2 -25040.5} C_VEL
LIN {X 0,Y 57.784,Z 733.261,A -85,B 0,C 180,E1 -25050.124,E2 -25050.124} C_VEL
LIN {X 0,Y 62.937,Z 731.136,A -85,B 0,C 180,E1 -25057.139,E2 -25057.139} C_VEL
LIN {X 0,Y 68.894,Z 729.264,A -85,B 0,C 180,E1 -25064.161,E2 -25064.161} C_VEL
LIN {X 0,Y 76.377,Z 726.496,A -85,B 0,C 180,E1 -25069.406,E2 -25069.406} C_VEL
LIN {X 0,Y 83.252,Z 724.561,A -85,B 0,C 180,E1 -25073.845,E2 -25073.845} C_VEL
LIN {X 0,Y 73.644,Z 734.549,A -85,B 0,C 180,E1 -25079.835,E2 -25079.835} C_VEL
LIN {X 0,Y 63.709,Z 743.748,A -85,B 0,C 180,E1 -25088.83,E2 -25088.83} C_VEL
LIN {X 0,Y 55.65,Z 750.771,A -85,B 0,C 180,E1 -25100.683,E2 -25100.683} C_VEL
LIN {X 0,Y 50.071,Z 756.343,A -85,B 0,C 180,E1 -25116.869,E2 -25116.869} C_VEL
LIN {X 0,Y 48.394,Z 759.667,A -85,B 0,C 180,E1 -25133.099,E2 -25133.099} C_VEL
LIN {X 0,Y 49.771,Z 761.695,A -85,B 0,C 180,E1 -25150.229,E2 -25150.229} C_VEL
LIN {X 0,Y 55.608,Z 762.328,A -85,B 0,C 180,E1 -25167.659,E2 -25167.659} C_VEL
LIN {X 0,Y 64.715,Z 761.262,A -85,B 0,C 180,E1 -25180.438,E2 -25180.438} C_VEL
LIN {X 0,Y 77.063,Z 758.174,A -85,B 0,C 180,E1 -25190.369,E2 -25190.369} C_VEL
LIN {X 0,Y 90.096,Z 753.471,A -85,B 0,C 180,E1 -25197.031,E2 -25197.031} C_VEL
LIN {X 0,Y 104.034,Z 746.718,A -85,B 0,C 180,E1 -25201.965,E2 -25201.965} C_VEL
LIN {X 0,Y 117.126,Z 738.685,A -85,B 0,C 180,E1 -25205.386,E2 -25205.386} C_VEL
LIN {X 0,Y 129.766,Z 728.943,A -85,B 0,C 180,E1 -25207.971,E2 -25207.971} C_VEL
LIN {X 0,Y 135.48,Z 723.816,A -85,B 0,C 180,E1 -25208.968,E2 -25208.968} C_VEL
LIN {X 0,Y 122.347,Z 734.863,A -85,B 0,C 180,E1 -25211.311,E2 -25211.311} C_VEL
LIN {X 0,Y 109.158,Z 744.014,A -85,B 0,C 180,E1 -25214.317,E2 -25214.317} C_VEL
LIN {X 0,Y 94.094,Z 752.431,A -85,B 0,C 180,E1 -25218.985,E2 -25218.985} C_VEL
LIN {X 0,Y 80.557,Z 758.406,A -85,B 0,C 180,E1 -25225.053,E2 -25225.053} C_VEL
LIN {X 0,Y 75.947,Z 760.138,A -85,B 0,C 180,E1 -25227.77,E2 -25227.77} C_VEL
LIN {X 0,Y 69.714,Z 762.031,A -85,B 0,C 180,E1 -25231.123,E2 -25231.123} C_VEL
LIN {X 0,Y 57.573,Z 764.469,A -85,B 0,C 180,E1 -25237.029,E2 -25237.029} C_VEL
LIN {X 0,Y 49.742,Z 765.445,A -85,B 0,C 180,E1 -25243.668,E2 -25243.668} C_VEL
LIN {X 0,Y 47.443,Z 765.646,A -85,B 0,C 180,E1 -25247.357,E2 -25247.357} C_VEL
LIN {X 0,Y 41.198,Z 765.581,A -85,B 0,C 180,E1 -25268.668,E2 -25268.668} C_VEL
LIN {X 0,Y 40.571,Z 764.124,A -85,B 0,C 180,E1 -25288.603,E2 -25288.603} C_VEL
LIN {X 0,Y 40.775,Z 761.817,A -85,B 0,C 180,E1 -25304.21,E2 -25304.21} C_VEL
LIN {X 0,Y 45.292,Z 756.771,A -85,B 0,C 180,E1 -25325.044,E2 -25325.044} C_VEL
LIN {X 0,Y 52.788,Z 750.756,A -85,B 0,C 180,E1 -25338.481,E2 -25338.481} C_VEL
LIN {X 0,Y 44.063,Z 744.166,A -85,B 0,C 180,E1 -25372.18,E2 -25372.18} C_VEL
LIN {X 0,Y 44.072,Z 743.062,A -85,B 0,C 180,E1 -25378.705,E2 -25378.705} C_VEL
LIN {X 0,Y 46.096,Z 740.44,A -85,B 0,C 180,E1 -25397.683,E2 -25397.683} C_VEL
LIN {X 0,Y 48.366,Z 739.221,A -85,B 0,C 180,E1 -25404.427,E2 -25404.427} C_VEL
LIN {X 0,Y 53.297,Z 737.436,A -85,B 0,C 180,E1 -25415.566,E2 -25415.566} C_VEL
LIN {X 0,Y 58.435,Z 735.657,A -85,B 0,C 180,E1 -25421.865,E2 -25421.865} C_VEL
LIN {X 0,Y 65.906,Z 733.598,A -85,B 0,C 180,E1 -25429.341,E2 -25429.341} C_VEL
LIN {X 0,Y 71.597,Z 731.764,A -85,B 0,C 180,E1 -25432.955,E2 -25432.955} C_VEL
LIN {X 0,Y 61.08,Z 741.123,A -85,B 0,C 180,E1 -25440.577,E2 -25440.577} C_VEL
LIN {X 0,Y 51.351,Z 748.855,A -85,B 0,C 180,E1 -25451.836,E2 -25451.836} C_VEL
LIN {X 0,Y 44.033,Z 754.84,A -85,B 0,C 180,E1 -25467.7,E2 -25467.7} C_VEL
LIN {X 0,Y 40.624,Z 758.925,A -85,B 0,C 180,E1 -25487.162,E2 -25487.162} C_VEL
LIN {X 0,Y 41.171,Z 761.455,A -85,B 0,C 180,E1 -25507.363,E2 -25507.363} C_VEL
LIN {X 0,Y 46.909,Z 762.746,A -85,B 0,C 180,E1 -25528.467,E2 -25528.467} C_VEL
LIN {X 0,Y 56.45,Z 762.234,A -85,B 0,C 180,E1 -25542.992,E2 -25542.992} C_VEL
LIN {X 0,Y 69.416,Z 759.848,A -85,B 0,C 180,E1 -25553.564,E2 -25553.564} C_VEL
LIN {X 0,Y 82.977,Z 755.82,A -85,B 0,C 180,E1 -25560.282,E2 -25560.282} C_VEL
LIN {X 0,Y 98.076,Z 749.511,A -85,B 0,C 180,E1 -25565.262,E2 -25565.262} C_VEL
LIN {X 0,Y 111.158,Z 742.379,A -85,B 0,C 180,E1 -25568.376,E2 -25568.376} C_VEL
LIN {X 0,Y 113.601,Z 740.829,A -85,B 0,C 180,E1 -25568.937,E2 -25568.937} C_VEL
LIN {X 0,Y 99.18,Z 749.152,A -85,B 0,C 180,E1 -25572.106,E2 -25572.106} C_VEL
LIN {X 0,Y 84.518,Z 755.857,A -85,B 0,C 180,E1 -25576.645,E2 -25576.645} C_VEL
LIN {X 0,Y 69.548,Z 761.078,A -85,B 0,C 180,E1 -25583.734,E2 -25583.734} C_VEL
LIN {X 0,Y 56.658,Z 764.252,A -85,B 0,C 180,E1 -25593.981,E2 -25593.981} C_VEL
LIN {X 0,Y 47.443,Z 765.646,A -85,B 0,C 180,E1 -25607.357,E2 -25607.357} C_VEL
LIN {X 0,Y 42.964,Z 765.79,A -85,B 0,C 180,E1 -25616.291,E2 -25616.291} C_VEL
LIN {X 0,Y 37.081,Z 765.186,A -85,B 0,C 180,E1 -25629.959,E2 -25629.959} C_VEL
LIN {X 0,Y 32.516,Z 762.639,A -85,B 0,C 180,E1 -25655.897,E2 -25655.897} C_VEL
LIN {X 0,Y 35.198,Z 758.703,A -85,B 0,C 180,E1 -25680.772,E2 -25680.772} C_VEL
LIN {X 0,Y 43.194,Z 752.736,A -85,B 0,C 180,E1 -25699.995,E2 -25699.995} C_VEL
LIN {X 0,Y 37.08,Z 746.957,A -85,B 0,C 180,E1 -25738.46,E2 -25738.46} C_VEL
LIN {X 0,Y 39.91,Z 744.302,A -85,B 0,C 180,E1 -25762.079,E2 -25762.079} C_VEL
LIN {X 0,Y 42.198,Z 743.321,A -85,B 0,C 180,E1 -25768.293,E2 -25768.293} C_VEL
LIN {X 0,Y 48.564,Z 741.49,A -85,B 0,C 180,E1 -25781.217,E2 -25781.217} C_VEL
LIN {X 0,Y 54.255,Z 739.826,A -85,B 0,C 180,E1 -25787.496,E2 -25787.496} C_VEL
LIN {X 0,Y 59.048,Z 738.776,A -85,B 0,C 180,E1 -25792.274,E2 -25792.274} C_VEL
LIN {X 0,Y 47.701,Z 747.243,A -85,B 0,C 180,E1 -25802.525,E2 -25802.525} C_VEL
LIN {X 0,Y 38.542,Z 753.625,A -85,B 0,C 180,E1 -25818.006,E2 -25818.006} C_VEL
LIN {X 0,Y 32.962,Z 758.553,A -85,B 0,C 180,E1 -25842.24,E2 -25842.24} C_VEL
LIN {X 0,Y 33.031,Z 761.417,A -85,B 0,C 180,E1 -25867.233,E2 -25867.233} C_VEL
LIN {X 0,Y 38.807,Z 762.993,A -85,B 0,C 180,E1 -25891.131,E2 -25891.131} C_VEL
LIN {X 0,Y 50.305,Z 762.877,A -85,B 0,C 180,E1 -25908.531,E2 -25908.531} C_VEL
LIN {X 0,Y 63.997,Z 760.922,A -85,B 0,C 180,E1 -25918.667,E2 -25918.667} C_VEL
LIN {X 0,Y 79.309,Z 756.962,A -85,B 0,C 180,E1 -25925.246,E2 -25925.246} C_VEL
LIN {X 0,Y 91.563,Z 752.466,A -85,B 0,C 180,E1 -25928.84,E2 -25928.84} C_VEL
LIN {X 0,Y 75.117,Z 758.616,A -85,B 0,C 180,E1 -25933.707,E2 -25933.707} C_VEL
LIN {X 0,Y 59.971,Z 762.654,A -85,B 0,C 180,E1 -25941.019,E2 -25941.019} C_VEL
LIN {X 0,Y 45.721,Z 764.96,A -85,B 0,C 180,E1 -25953.822,E2 -25953.822} C_VEL
LIN {X 0,Y 35.845,Z 765.359,A -85,B 0,C 180,E1 -25974.165,E2 -25974.165} C_VEL
LIN {X 0,Y 32.426,Z 764.054,A -85,B 0,C 180,E1 -26001.151,E2 -26001.151} C_VEL
LIN {X 0,Y 32.576,Z 763.11,A -85,B 0,C 180,E1 -26011.778,E2 -26011.778} C_VEL
LIN {X 0,Y 32.516,Z 762.639,A -85,B 0,C 180,E1 -26015.897,E2 -26015.897} C_VEL
LIN {X 0,Y 31.778,Z 761.477,A -85,B 0,C 180,E1 -26024.885,E2 -26024.885} C_VEL
LIN {X 0,Y 29.954,Z 757.42,A -85,B 0,C 180,E1 -26050.738,E2 -26050.738} C_VEL
LIN {X 0,Y 31.735,Z 755.808,A -85,B 0,C 180,E1 -26057.838,E2 -26057.838} C_VEL
LIN {X 0,Y 33.735,Z 754.554,A -85,B 0,C 180,E1 -26062.001,E2 -26062.001} C_VEL
LIN {X 0,Y 29.833,Z 750.319,A -85,B 0,C 180,E1 -26100.007,E2 -26100.007} C_VEL
LIN {X 0,Y 33.883,Z 747.818,A -85,B 0,C 180,E1 -26128.181,E2 -26128.181} C_VEL
LIN {X 0,Y 36.59,Z 746.95,A -85,B 0,C 180,E1 -26135.026,E2 -26135.026} C_VEL
LIN {X 0,Y 45.04,Z 745.008,A -85,B 0,C 180,E1 -26149.013,E2 -26149.013} C_VEL
LIN {X 0,Y 46.78,Z 744.592,A -85,B 0,C 180,E1 -26150.894,E2 -26150.894} C_VEL
LIN {X 0,Y 35.742,Z 751.501,A -85,B 0,C 180,E1 -26163.392,E2 -26163.392} C_VEL
LIN {X 0,Y 26.735,Z 757.193,A -85,B 0,C 180,E1 -26187.833,E2 -26187.833} C_VEL
LIN {X 0,Y 24.458,Z 760.653,A -85,B 0,C 180,E1 -26219.348,E2 -26219.348} C_VEL
LIN {X 0,Y 29.577,Z 762.918,A -85,B 0,C 180,E1 -26251.745,E2 -26251.745} C_VEL
LIN {X 0,Y 41.36,Z 763.573,A -85,B 0,C 180,E1 -26272.256,E2 -26272.256} C_VEL
LIN {X 0,Y 55.037,Z 762.536,A -85,B 0,C 180,E1 -26282.597,E2 -26282.597} C_VEL
LIN {X 0,Y 69.552,Z 759.824,A -85,B 0,C 180,E1 -26288.675,E2 -26288.675} C_VEL
LIN {X 0,Y 53.884,Z 763.191,A -85,B 0,C 180,E1 -26295.271,E2 -26295.271} C_VEL
LIN {X 0,Y 38.52,Z 764.842,A -85,B 0,C 180,E1 -26308.085,E2 -26308.085} C_VEL
LIN {X 0,Y 27.583,Z 764.667,A -85,B 0,C 180,E1 -26331.987,E2 -26331.987} C_VEL
LIN {X 0,Y 24.516,Z 762.987,A -85,B 0,C 180,E1 -26365.347,E2 -26365.347} C_VEL
LIN {X 0,Y 24.53,Z 762.012,A -85,B 0,C 180,E1 -26377.049,E2 -26377.049} C_VEL
LIN {X 0,Y 28.553,Z 757.803,A -85,B 0,C 180,E1 -26409.1,E2 -26409.1} C_VEL
LIN {X 0,Y 31.735,Z 755.808,A -85,B 0,C 180,E1 -26417.838,E2 -26417.838} C_VEL
LIN {X 0,Y 32.189,Z 754.973,A -85,B 0,C 180,E1 -26421.676,E2 -26421.676} C_VEL
LIN {X 0,Y 31.17,Z 754.229,A -85,B 0,C 180,E1 -26427.081,E2 -26427.081} C_VEL
LIN {X 0,Y 28.419,Z 753.723,A -85,B 0,C 180,E1 -26435.146,E2 -26435.146} C_VEL
LIN {X 0,Y 22.653,Z 753.395,A -85,B 0,C 180,E1 -26459.414,E2 -26459.414} C_VEL
LIN {X 0,Y 22.534,Z 753.135,A -85,B 0,C 180,E1 -26466.427,E2 -26466.427} C_VEL
